// §6.8 ST step skeleton. One M_Step per step, one commit via M_Advance.
METHOD M_ChainRun
IF NOT _attached THEN
    RETURN;
END_IF
CASE _step OF
    0:  // ram up
        M_Step(StepNo := _baseStepNo, StepName := 'project.step.pressSafePositionRamUp',
            Awaits := _pressRam, AwaitingLabel := 'PressRam.RETRACT',
            TimeClass := E_TimeClass.WORK, ExpectedTime := T#0S, Branch := 0);
        IF M_TryIssue(Steppable := TRUE) THEN
            _pressRam.Abort := FALSE;
            _pressRam.Command := E_CylinderCommand.RETRACT;
            _pressRam.Execute := TRUE;
        END_IF
        IF _pressRam.Done THEN
            _pressRam.Execute := FALSE;
            _retVal := E_StepResult.ADVANCE;
        END_IF
        M_Advance(OnAdvance := 20, OnJump1 := -1, OnJump2 := -1, OnJump3 := -1);
    20:  // door open
        M_Step(StepNo := _baseStepNo + 20, StepName := 'project.step.pressSafePositionDoorOpen',
            Awaits := _door, AwaitingLabel := 'Door.RETRACT',
            TimeClass := E_TimeClass.WORK, ExpectedTime := T#0S, Branch := 0);
        IF M_TryIssue(Steppable := TRUE) THEN
            _door.Abort := FALSE;
            _door.Command := E_CylinderCommand.RETRACT;
            _door.Execute := TRUE;
        END_IF
        IF _door.Done THEN
            _door.Execute := FALSE;
            _retVal := E_StepResult.ADVANCE;
        END_IF
        M_Advance(OnAdvance := 40, OnJump1 := -1, OnJump2 := -1, OnJump3 := -1);
    40:  // slide outside
        M_Step(StepNo := _baseStepNo + 40, StepName := 'project.step.pressSafePositionSlideOutside',
            Awaits := _partSlide, AwaitingLabel := 'PartSlide.RETRACT',
            TimeClass := E_TimeClass.WORK, ExpectedTime := T#0S, Branch := 0);
        IF M_TryIssue(Steppable := TRUE) THEN
            _partSlide.Abort := FALSE;
            _partSlide.Command := E_CylinderCommand.RETRACT;
            _partSlide.Execute := TRUE;
        END_IF
        IF _partSlide.Done THEN
            _partSlide.Execute := FALSE;
            _retVal := E_StepResult.ADVANCE;
        END_IF
        M_Advance(OnAdvance := 999, OnJump1 := -1, OnJump2 := -1, OnJump3 := -1);
    999:  // established
        M_Step(StepNo := _baseStepNo + 60, StepName := 'project.step.pressSafePositionComplete',
            Awaits := 0, AwaitingLabel := '', TimeClass := E_TimeClass.WORK, ExpectedTime := T#0S, Branch := 0);
        Done := TRUE;
ELSE
    M_Fault(Reason := E_Reason.STEP_STALLED, DescriptionKey := 'std.error.undefinedStep');
END_CASE
END_METHOD

METHOD Setup : BOOL
VAR_INPUT
    Host : I_SequenceHost;
END_VAR
VAR_IN_OUT
    PressRam : FB_CylinderCM;
    Door : FB_CylinderCM;
    PartSlide : FB_CylinderCM;
END_VAR
_pressRam REF= PressRam;
_door REF= Door;
_partSlide REF= PartSlide;
Setup := M_Attach(Host := Host)
    AND __ISVALIDREF(_pressRam) AND __ISVALIDREF(_door) AND __ISVALIDREF(_partSlide);
END_METHOD

END_FUNCTION_BLOCK

// ---- 01_PneumaticPress/Sequences/FB_PressDemoChangeover.TcPOU
// CHANGEOVER mode chain (Core §6.2/§6.8 ST skeleton on FB_SequenceBase): validate
// the selected model, establish the shared load-safe position, then ask the
// operator (§6.11) to confirm tooling/material match before completing. The
// 'repeat position' answer restarts the guided move via a backward jump (§6.10).
FUNCTION_BLOCK FB_PressDemoChangeover EXTENDS FB_SequenceBase
VAR
    _decisionRequest : ST_DecisionRequest;
    _answer : INT;
    _modelSelected : BOOL;
    {attribute 'OPC.UA.DA' := '0'}
    _outCmd : REFERENCE TO ST_PneumaticPressOutCmd;
    {attribute 'OPC.UA.DA' := '0'}
    _model : REFERENCE TO ST_ModelId;
    {attribute 'OPC.UA.DA' := '0'}
    _loadPosition : FB_PressDemoLoadPosition;
END_VAR

// §6.8 - the chain's own state on a restart (the base resets the flow state).
METHOD PROTECTED OnChainReset
_answer := 0;
END_METHOD

METHOD M_Run
IF NOT _attached THEN
    RETURN;
END_IF
CASE _step OF
    0:  // initialize
        M_Step(StepNo := 0, StepName := 'project.step.pressChangeoverInitialize',
            Awaits := 0, AwaitingLabel := '', TimeClass := E_TimeClass.WORK, ExpectedTime := T#0S, Branch := 0);
        _outCmd.ChangeoverCompleted := FALSE;
        _answer := 0;
        _decisionRequest.Prompt := '';
        M_ClearDecision();
        _retVal := E_StepResult.ADVANCE;
        M_Advance(OnAdvance := 800, OnJump1 := -1, OnJump2 := -1, OnJump3 := -1);
    800:  // validate the transactionally-loaded model
        M_Step(StepNo := 800, StepName := 'project.step.pressChangeoverValidateModel',
            Awaits := 0, AwaitingLabel := '', TimeClass := E_TimeClass.WAIT_OPERATOR, ExpectedTime := T#0S, Branch := 0);
        _modelSelected := M_Await(Idx := 1, Label := 'project.condition.pressModelSelected',
            Ok := _model.ModelCode <> '');
        IF _modelSelected THEN
            _retVal := E_StepResult.ADVANCE;
        END_IF
        M_Advance(OnAdvance := 810, OnJump1 := -1, OnJump2 := -1, OnJump3 := -1);
    810:  // shared load-safe position (composite step)
        _retVal := M_RunSub(Chain := _loadPosition, BaseStepNo := 810);
        M_Advance(OnAdvance := 870, OnJump1 := -1, OnJump2 := -1, OnJump3 := -1);
    870:  // request tooling/material confirmation
        M_Step(StepNo := 870, StepName := 'project.step.pressChangeoverRequestConfirmation',
            Awaits := 0, AwaitingLabel := '', TimeClass := E_TimeClass.WAIT_OPERATOR, ExpectedTime := T#0S, Branch := 0);
        _decisionRequest.Prompt := 'project.decision.pressChangeoverConfirm';
        _decisionRequest.Options[1] := 'project.decision.confirmChangeover';
        _decisionRequest.Options[2] := 'project.decision.repeatChangeoverPosition';
        _decisionRequest.Default := 0;
        _decisionRequest.Timeout := T#0S;
        M_AskDecision(Req := _decisionRequest);
        _retVal := E_StepResult.ADVANCE;
        M_Advance(OnAdvance := 880, OnJump1 := -1, OnJump2 := -1, OnJump3 := -1);
    880:  // await confirmation; JUMP1 = repeat the guided position
        M_Step(StepNo := 880, StepName := 'project.step.pressChangeoverAwaitConfirmation',
            Awaits := 0, AwaitingLabel := '', TimeClass := E_TimeClass.WAIT_OPERATOR, ExpectedTime := T#0S, Branch := 0);
        _answer := M_TakeDecision();
        IF _answer = 1 THEN
            _retVal := E_StepResult.ADVANCE;
        ELSIF _answer = 2 THEN
            _retVal := E_StepResult.JUMP1;
        ELSE
            _modelSelected := M_Await(Idx := 1,
                Label := 'project.condition.pressChangeoverConfirmation', Ok := FALSE);
        END_IF
        M_Advance(OnAdvance := 999, OnJump1 := 810, OnJump2 := -1, OnJump3 := -1);
    999:  // complete
        M_Step(StepNo := 999, StepName := 'project.step.pressChangeoverComplete',
            Awaits := 0, AwaitingLabel := '', TimeClass := E_TimeClass.WORK, ExpectedTime := T#0S, Branch := 0);
        _outCmd.ChangeoverCompleted := TRUE;
        M_Complete();
ELSE
    M_Fault(Reason := E_Reason.STEP_STALLED, DescriptionKey := 'std.error.undefinedStep');
END_CASE
END_METHOD

METHOD Setup : BOOL
VAR_INPUT
    Host : I_SequenceHost;
END_VAR
VAR_IN_OUT
    PressRam : FB_CylinderCM;
    Door : FB_CylinderCM;
    PartSlide : FB_CylinderCM;
    OutCmd : ST_PneumaticPressOutCmd;
    Model : ST_ModelId;
END_VAR
_outCmd REF= OutCmd;
_model REF= Model;
Setup := M_Attach(Host := Host) AND __ISVALIDREF(_outCmd) AND __ISVALIDREF(_model)
    AND _loadPosition.Setup(Host := Host, PressRam := PressRam, Door := Door, PartSlide := PartSlide);
END_METHOD

END_FUNCTION_BLOCK

// ---- 01_PneumaticPress/Sequences/FB_PressDemoAuto.TcPOU
// AUTO mode chain (Core §6.2/§6.8 ST skeleton on FB_SequenceBase): the continuous
// production cycle — await a fresh two-hand start with part+air present, transfer
// the part in, press for the recipe dwell, return to load position, count the good
// part, and loop until Stop. A Stop requested at the between-cycles wait is honored
// there (M_StopNow) so no phantom cycle is charged. Every child motion goes through
// the §6.1 handshake (M_TryIssue); progression rides the shared _retVal.
FUNCTION_BLOCK FB_PressDemoAuto EXTENDS FB_SequenceBase
VAR
    _partReady, _airReady, _startReady : BOOL;
    _dwellTwoHandHeld : BOOL;          // N220 named wait: two-hand held through the dwell
    _decisionRequest : ST_DecisionRequest;   // §6.11 not-reached confirmation
    _answer : INT;
    _ramReached, _failureConfirmed : BOOL;   // N200/N210 named waits
    _twoHandHeldDuringClose : BOOL;          // N180 named wait
    _closeAbortWarned : BOOL;                // N180 §6.9(e) message result
    _ramFailureReported : BOOL;              // N200 §6.9(e) message result
    _partInMachine : BOOL;                   // §3.16.3 the part is already received
    _partDispositioned : BOOL;               // N260 already set the verdict
    _traceAccepted, _recordAccepted, _partProcessed : BOOL;
    {attribute 'OPC.UA.DA' := '0'}
    _pressRam : REFERENCE TO FB_CylinderCM;
    {attribute 'OPC.UA.DA' := '0'}
    _door : REFERENCE TO FB_CylinderCM;
    {attribute 'OPC.UA.DA' := '0'}
    _partSlide : REFERENCE TO FB_CylinderCM;
    {attribute 'OPC.UA.DA' := '0'}
    _twoHand : REFERENCE TO FB_TwoHandStartCM;
    {attribute 'OPC.UA.DA' := '0'}
    _partPresentSensor : REFERENCE TO FB_DigitalInputCM;
    {attribute 'OPC.UA.DA' := '0'}
    _airPressureMonitor : REFERENCE TO FB_AirPressureMonitorCM;
    {attribute 'OPC.UA.DA' := '0'}
    _parCfg : REFERENCE TO ST_PneumaticPressParCfg;
    // §3.8a - the CELL's own policy, held separately from the MODEL's data and
    // referenced exactly like _parCfg, so each step reads whichever structure
    // actually owns the value it is asking about.
    {attribute 'OPC.UA.DA' := '0'}
    _stationCfg : REFERENCE TO ST_PneumaticPressStationCfg;
    {attribute 'OPC.UA.DA' := '0'}
    _outCmd : REFERENCE TO ST_PneumaticPressOutCmd;
    {attribute 'OPC.UA.DA' := '0'}
    _startLatched : REFERENCE TO BOOL;
    {attribute 'OPC.UA.DA' := '0'}
    _loadPosition : FB_PressDemoLoadPosition;
END_VAR

// §6.8 - the chain's own state on a restart (the base resets the flow state).
METHOD PROTECTED OnChainReset
// A chart restart abandons whatever the cycle was holding: the part record is
// closed by N215/N999, never by a restart, so both trackers start clean.
_partDispositioned := FALSE;
_partInMachine := FALSE;
END_METHOD

METHOD M_Run
IF NOT _attached THEN
    RETURN;
END_IF
CASE _step OF
    0:  // initialize
        M_Step(StepNo := 0, StepName := 'project.step.pressAutoInitialize',
            Awaits := 0, AwaitingLabel := '', TimeClass := E_TimeClass.WORK, ExpectedTime := T#0S, Branch := 0);
        _outCmd.CycleCompleted := FALSE;
        _retVal := E_StepResult.ADVANCE;
        M_Advance(OnAdvance := 100, OnJump1 := -1, OnJump2 := -1, OnJump3 := -1 );
    100:  // await a fresh two-hand start (the §8.11.1 cycle-start marker)
        M_Step(StepNo := 100, StepName := 'project.step.pressAwaitTwoHand',
            Awaits := 0, AwaitingLabel := '', TimeClass := E_TimeClass.WAIT_OPERATOR, ExpectedTime := T#0S, Branch := 0);
        _outCmd.CycleCompleted := FALSE;
        _partReady := M_Await(Idx := 1, Label := 'project.condition.partPresent',
            Ok := _partPresentSensor.OutImm.Value AND _partPresentSensor.OutImm.Quality);
        _airReady := M_Await(Idx := 2, Label := 'project.condition.airPressureOk',
            Ok := _airPressureMonitor.OutImm.PressureOk);
        IF _stationCfg.RequireTwoHandStart THEN
            _startReady := M_Await(Idx := 3, Label := 'project.condition.twoHandStart', Ok := _startLatched);
        ELSE
            _startReady := TRUE;
        END_IF
        IF M_StopPending() THEN
            M_StopNow();                       // stop accepted BETWEEN cycles: no phantom cycle
        ELSIF _partReady AND _airReady AND _startReady THEN
            // §3.16.3 receive once per PHYSICAL part. The N180 two-hand abort returns
            // here with the same part still in the machine and nothing processed, so a
            // second M_PartReceived would open a duplicate record for one part.
            // M_PartStarted (N150) is deliberately NOT guarded: each pass is a genuine
            // processing attempt on that part.
            IF NOT _partInMachine THEN
                _traceAccepted := M_PartReceived();
                _partInMachine := TRUE;
            END_IF
            _retVal := E_StepResult.ADVANCE;
        END_IF
        M_Advance(OnAdvance := 110, OnJump1 := -1, OnJump2 := -1, OnJump3 := -1);
    110:  // ram up
        M_Step(StepNo := 110, StepName := 'project.step.pressRamUp',
            Awaits := _pressRam, AwaitingLabel := 'PressRam.RETRACT', TimeClass := E_TimeClass.WORK, ExpectedTime := T#0S, Branch := 0);
        IF M_TryIssue(Steppable := TRUE) THEN
            _pressRam.Abort := FALSE; _pressRam.Command := E_CylinderCommand.RETRACT; _pressRam.Execute := TRUE;
        END_IF
        IF _pressRam.Done THEN _pressRam.Execute := FALSE; _retVal := E_StepResult.ADVANCE; END_IF
        M_Advance(OnAdvance := 130, OnJump1 := -1, OnJump2 := -1, OnJump3 := -1);
    130:  // door open
        M_Step(StepNo := 130, StepName := 'project.step.pressDoorOpen',
            Awaits := _door, AwaitingLabel := 'Door.RETRACT', TimeClass := E_TimeClass.WORK, ExpectedTime := T#0S, Branch := 0);
        IF M_TryIssue(Steppable := TRUE) THEN
            _door.Abort := FALSE; _door.Command := E_CylinderCommand.RETRACT; _door.Execute := TRUE;
        END_IF
        IF _door.Done THEN _door.Execute := FALSE; _retVal := E_StepResult.ADVANCE; END_IF
        M_Advance(OnAdvance := 150, OnJump1 := -1, OnJump2 := -1, OnJump3 := -1);
    150:  // slide inside (value-adding sequence begins)
        M_Step(StepNo := 150, StepName := 'project.step.pressSlideInside',
            Awaits := _partSlide, AwaitingLabel := 'PartSlide.EXTEND', TimeClass := E_TimeClass.WORK, ExpectedTime := T#0S, Branch := 0);
        IF M_TryIssue(Steppable := TRUE) THEN
            M_PartStarted();
            _partSlide.Abort := FALSE; _partSlide.Command := E_CylinderCommand.EXTEND; _partSlide.Execute := TRUE;
        END_IF
        IF _partSlide.Done THEN _partSlide.Execute := FALSE; _retVal := E_StepResult.ADVANCE; END_IF
        M_Advance(OnAdvance := 170, OnJump1 := -1, OnJump2 := -1, OnJump3 := -1);
    170:  // transfer settle
        M_Step(StepNo := 170, StepName := 'project.step.pressTransferSettle',
            Awaits := 0, AwaitingLabel := '', TimeClass := E_TimeClass.WORK, ExpectedTime := _parCfg.TransferSettleTime, Branch := 0);
        _retVal := M_Delay(PT := _parCfg.TransferSettleTime);
        M_Advance(OnAdvance := 180, OnJump1 := -1, OnJump2 := -1, OnJump3 := -1);
    180:  // door close. Releasing a two-hand button while the door is moving is an
          // operator abort, not a fault: the door goes back up, the part slides out,
          // and the cycle returns to the two-hand wait (§6.10 jump). Completion wins
          // if the door finished in the same scan the button was released.
        M_Step(StepNo := 180, StepName := 'project.step.pressDoorClose',
            Awaits := _door, AwaitingLabel := 'Door.EXTEND', TimeClass := E_TimeClass.WORK, ExpectedTime := T#0S, Branch := 0);
        _twoHandHeldDuringClose := M_Await(Idx := 1,
            Label := 'project.condition.twoHandHeldDuringDoorClose',
            Ok := _twoHand.OutImm.SafeActive OR NOT _stationCfg.RequireTwoHandStart);
        IF M_TryIssue(Steppable := TRUE) THEN
            _door.Abort := FALSE; _door.Command := E_CylinderCommand.EXTEND; _door.Execute := TRUE;
        END_IF
        IF _door.Done THEN
            _door.Execute := FALSE;
            _retVal := E_StepResult.ADVANCE;
        ELSIF NOT _twoHandHeldDuringClose THEN
            _door.Execute := FALSE;             // §6.1 Execute-drop reset releases the close
            // §6.9(e) — a WARNING, not a fault: the release is designed operator
            // behaviour and the chain already owns the recovery below, so nothing
            // stops. It is recorded because a cycle was abandoned with the part
            // still in the machine, and the §3.13 chart marks this step for it.
            // The base raises it once per visit however many scans this runs.
            _closeAbortWarned := M_RaiseWarning(
                Reason := PL_PressReasons.PRESS_TWO_HAND_RELEASED,
                DescriptionKey := 'project.warning.twoHandReleasedDuringDoorClose',
                Severity := E_Severity.LOW, Category := E_Category.PROCESS);
            _retVal := E_StepResult.JUMP1;      // released -> reopen and clear the part
        END_IF
        M_Advance(OnAdvance := 200, OnJump1 := 185, OnJump2 := -1, OnJump3 := -1);
    185:  // two-hand released during closing: take the door back up
        M_Step(StepNo := 185, StepName := 'project.step.pressDoorReopen',
            Awaits := _door, AwaitingLabel := 'Door.RETRACT', TimeClass := E_TimeClass.WORK, ExpectedTime := T#0S, Branch := 0);
        IF M_TryIssue(Steppable := TRUE) THEN
            _door.Abort := FALSE; _door.Command := E_CylinderCommand.RETRACT; _door.Execute := TRUE;
        END_IF
        IF _door.Done THEN _door.Execute := FALSE; _retVal := E_StepResult.ADVANCE; END_IF
        M_Advance(OnAdvance := 190, OnJump1 := -1, OnJump2 := -1, OnJump3 := -1);
    190:  // slide the part back out, then return to the two-hand wait. The start latch
          // is dropped so the cycle cannot resume without a fresh two-hand press.
        M_Step(StepNo := 190, StepName := 'project.step.pressSlideOutsideAfterAbort',
            Awaits := _partSlide, AwaitingLabel := 'PartSlide.RETRACT', TimeClass := E_TimeClass.WORK, ExpectedTime := T#0S, Branch := 0);
        IF M_TryIssue(Steppable := TRUE) THEN
            _partSlide.Abort := FALSE; _partSlide.Command := E_CylinderCommand.RETRACT; _partSlide.Execute := TRUE;
        END_IF
        IF _partSlide.Done THEN
            _partSlide.Execute := FALSE;
            _startLatched := FALSE;
            _retVal := E_StepResult.ADVANCE;
        END_IF
        M_Advance(OnAdvance := 100, OnJump1 := -1, OnJump2 := -1, OnJump3 := -1);
    200:  // ram down. THIS step owns the not-reached disposition, so it does NOT hand
          // the ram to the §6.9 auto-rollup: an awaited child fault is adopted by the
          // Unit (ERROR, _step := 0) before _M_Dispatch runs, and the chain would stop
          // before it could ask the operator anything. The wait is still named (§6.9(b))
          // and the cylinder still raises its own CYL_NOT_EXTENDED alarm.
        M_Step(StepNo := 200, StepName := 'project.step.pressRamDown',
            Awaits := 0, AwaitingLabel := '', TimeClass := E_TimeClass.WORK, ExpectedTime := T#0S, Branch := 0);
        _ramReached := M_Await(Idx := 1, Label := 'project.condition.pressRamExtended',
            Ok := _pressRam.Done);
        IF M_TryIssue(Steppable := TRUE) THEN
            _pressRam.Abort := FALSE; _pressRam.Command := E_CylinderCommand.EXTEND; _pressRam.Execute := TRUE;
        END_IF
        IF _pressRam.Done THEN
            _pressRam.Execute := FALSE;
            _retVal := E_StepResult.ADVANCE;
        ELSIF _pressRam.Error THEN
            // §6.9(e) — publish the ram's own first-out (CYL_NOT_EXTENDED, with its
            // text and IO tag) on the Unit and on this row of the §3.13 chart, and
            // do NOT adopt it: the confirmation + scrap below IS the handling, so a
            // fault here would replace a designed recovery. Saying nothing is what
            // left the failure visible only on the ram itself.
            _ramFailureReported := M_ReportFromChild(Source := _pressRam);
            _pressRam.Execute := FALSE;         // §6.1 Execute-drop reset returns the ram to READY
            _retVal := E_StepResult.JUMP1;      // did not reach -> operator confirmation
        END_IF
        M_Advance(OnAdvance := 220, OnJump1 := 210, OnJump2 := -1, OnJump3 := -1);
    210:  // press did not reach: the operator confirms the failure before the part is
          // scrapped. A scrap is deliberate, so there is no timeout default (§6.11).
        M_Step(StepNo := 210, StepName := 'project.step.pressNotReachedConfirm',
            Awaits := 0, AwaitingLabel := '', TimeClass := E_TimeClass.WAIT_OPERATOR, ExpectedTime := T#0S, Branch := 0);
        _decisionRequest.Prompt := 'project.decision.pressNotReached';
        _decisionRequest.Options[1] := 'project.decision.confirmScrapAndReturn';
        _decisionRequest.Default := 0;
        _decisionRequest.Timeout := T#0S;
        M_AskDecision(Req := _decisionRequest);
        _answer := M_TakeDecision();
        IF _answer = 1 THEN
            _retVal := E_StepResult.ADVANCE;
        ELSE
            _failureConfirmed := M_Await(Idx := 1,
                Label := 'project.condition.pressFailureConfirmation', Ok := FALSE);
        END_IF
        M_Advance(OnAdvance := 215, OnJump1 := -1, OnJump2 := -1, OnJump3 := -1);
    215:  // disposition the part NOK, then rejoin the shared return-to-start step
        M_Step(StepNo := 215, StepName := 'project.step.pressScrapPart',
            Awaits := 0, AwaitingLabel := '', TimeClass := E_TimeClass.WORK, ExpectedTime := T#0S, Branch := 0);
        _partProcessed := M_PartProcessed(Verdict := E_Verdict.NOK,
            Reason := PL_ModuleReasons.CYL_NOT_EXTENDED);
        _partDispositioned := TRUE;             // N999 must not also count it good
        _partInMachine := FALSE;                // dispositioned: the next one is a new part
        _outCmd.CycleCompleted := FALSE;
        _retVal := E_StepResult.ADVANCE;
        M_Advance(OnAdvance := 240, OnJump1 := -1, OnJump2 := -1, OnJump3 := -1);
    220:  // press dwell — two-hand must stay held; releasing it HOLDS the dwell
        M_Step(StepNo := 220, StepName := 'project.step.pressDwell',
            Awaits := 0, AwaitingLabel := '', TimeClass := E_TimeClass.WORK, ExpectedTime := _parCfg.PressSettleTime, Branch := 0);
        // Releasing the button mid-dwell is the designed way to stop pressing, so it
        // is a named wait (§6.9(b)), not a fault: the ram's outputs come off, the
        // dwell timer freezes where it is because M_Delay is not called, and pressing
        // again restores the force and finishes the remaining dwell. Faulting here
        // charged an unrecoverable downtime event for normal operator behaviour.
        _dwellTwoHandHeld := M_Await(Idx := 1, Label := 'project.condition.twoHandHeldDuringPress',
            Ok := _twoHand.OutImm.SafeActive OR NOT _stationCfg.RequireTwoHandStart);
        IF NOT _dwellTwoHandHeld THEN
            _pressRam.WithdrawOutputs();
        ELSE
            // The press force is the valve latched by the EXTEND that step 200 already
            // completed, so after a withdraw only this call re-energizes it — and the
            // ram re-checks its own extend permit before it does (§7.2).
            _pressRam.RestoreOutputs();
            _retVal := M_Delay(PT := _parCfg.PressSettleTime);
        END_IF
        M_Advance(OnAdvance := 230, OnJump1 := -1, OnJump2 := -1, OnJump3 := -1);
    230:  // record the applied dwell (§3.16.1 measured value)
        M_Step(StepNo := 230, StepName := 'project.step.pressRecordResult',
            Awaits := 0, AwaitingLabel := '', TimeClass := E_TimeClass.WORK, ExpectedTime := T#0S, Branch := 0);
        _recordAccepted := M_PartRecord(RecordName := 'PressDwell',
            Value := DINT_TO_LREAL(TIME_TO_DINT(_parCfg.PressSettleTime)),
            Minimum := 0, Maximum := 30000,
            Target := DINT_TO_LREAL(TIME_TO_DINT(_parCfg.PressSettleTime)), EngUnit := 'ms');
        _retVal := E_StepResult.ADVANCE;
        M_Advance(OnAdvance := 240, OnJump1 := -1, OnJump2 := -1, OnJump3 := -1);
    240:  // return to the shared load-safe position (composite step)
        _retVal := M_RunSub(Chain := _loadPosition, BaseStepNo := 240);
        M_Advance(OnAdvance := 999, OnJump1 := -1, OnJump2 := -1, OnJump3 := -1);
    999:  // cycle complete — write result, count by verdict, loop (§8.11.1 finish marker)
        M_Step(StepNo := 999, StepName := 'project.step.pressAutoComplete',
            Awaits := 0, AwaitingLabel := '', TimeClass := E_TimeClass.WORK, ExpectedTime := T#0S, Branch := 0);
        _outCmd.CycleCompleted := TRUE;
        IF _partDispositioned THEN
            _partDispositioned := FALSE;       // N260 already set the NOK verdict
        ELSE
            _partProcessed := M_PartProcessed(Verdict := E_Verdict.OK, Reason := E_Reason.NONE);
            IF NOT _partProcessed THEN
                M_CountGood();                 // §3.9: no carrier configured — count directly
            END_IF
        END_IF
        _partInMachine := FALSE;               // processed: the next one is a new part
        _startLatched := FALSE;
        IF M_EndOfCycle() THEN
            _retVal := E_StepResult.ADVANCE;   // stop NOT requested: loop to N100
        END_IF
        M_Advance(OnAdvance := 100, OnJump1 := -1, OnJump2 := -1, OnJump3 := -1);
ELSE
    M_Fault(Reason := E_Reason.STEP_STALLED, DescriptionKey := 'std.error.undefinedStep');
END_CASE
END_METHOD

METHOD Setup : BOOL
VAR_INPUT
    Host : I_SequenceHost;
END_VAR
VAR_IN_OUT
    PressRam : FB_CylinderCM;
    Door : FB_CylinderCM;
    PartSlide : FB_CylinderCM;
    TwoHand : FB_TwoHandStartCM;
    PartPresentSensor : FB_DigitalInputCM;
    AirPressureMonitor : FB_AirPressureMonitorCM;
    ParCfg : ST_PneumaticPressParCfg;
    StationCfg : ST_PneumaticPressStationCfg;
    OutCmd : ST_PneumaticPressOutCmd;
    StartLatched : BOOL;
END_VAR
_pressRam REF= PressRam;
_door REF= Door;
_partSlide REF= PartSlide;
_twoHand REF= TwoHand;
_partPresentSensor REF= PartPresentSensor;
_airPressureMonitor REF= AirPressureMonitor;
_parCfg REF= ParCfg;
_stationCfg REF= StationCfg;
_outCmd REF= OutCmd;
_startLatched REF= StartLatched;
Setup := M_Attach(Host := Host) AND __ISVALIDREF(_pressRam) AND __ISVALIDREF(_door)
    AND __ISVALIDREF(_partSlide) AND __ISVALIDREF(_twoHand)
    AND __ISVALIDREF(_partPresentSensor) AND __ISVALIDREF(_airPressureMonitor)
    AND __ISVALIDREF(_parCfg) AND __ISVALIDREF(_outCmd) AND __ISVALIDREF(_startLatched)
    AND _loadPosition.Setup(Host := Host, PressRam := PressRam, Door := Door, PartSlide := PartSlide);
END_METHOD

END_FUNCTION_BLOCK

// ---- 01_PneumaticPress/Sequences/FB_SFC_PressDemoAuto.TcPOU
// SFC rendition of FB_PressDemoAuto - identical behaviour, chart-language
// transitions. Every step action below sets the shared `_retVal`; the chart's
// transitions read it, and the owner calls M_BeginScan() once per PLC cycle
// before executing this chart so the result cannot survive into the next scan
// (Core §6.8). The ST twin remains FB_PressDemoAuto; keep the two in step.
FUNCTION_BLOCK INTERNAL FB_SFC_PressDemoAuto EXTENDS FB_SequenceBase
VAR
    _partReady, _airReady, _startReady : BOOL;
    _dwellTwoHandHeld : BOOL;          // N220 named wait: two-hand held through the dwell
    _decisionRequest : ST_DecisionRequest;   // §6.11 not-reached confirmation
    _answer : INT;
    _ramReached, _failureConfirmed : BOOL;   // N200/N210 named waits
    _twoHandHeldDuringClose : BOOL;
    _closeAbortWarned : BOOL;                // N180 §6.9(e) message result
    _ramFailureReported : BOOL;              // N200 §6.9(e) message result          // N180 named wait
    _partInMachine : BOOL;                   // §3.16.3 the part is already received
    _partDispositioned : BOOL;               // N260 already set the verdict
    _traceAccepted, _recordAccepted, _partProcessed : BOOL;
    {attribute 'OPC.UA.DA' := '0'}
    _pressRam : REFERENCE TO FB_CylinderCM;
    {attribute 'OPC.UA.DA' := '0'}
    _door : REFERENCE TO FB_CylinderCM;
    {attribute 'OPC.UA.DA' := '0'}
    _partSlide : REFERENCE TO FB_CylinderCM;
    {attribute 'OPC.UA.DA' := '0'}
    _twoHand : REFERENCE TO FB_TwoHandStartCM;
    {attribute 'OPC.UA.DA' := '0'}
    _partPresentSensor : REFERENCE TO FB_DigitalInputCM;
    {attribute 'OPC.UA.DA' := '0'}
    _airPressureMonitor : REFERENCE TO FB_AirPressureMonitorCM;
    {attribute 'OPC.UA.DA' := '0'}
    _parCfg : REFERENCE TO ST_PneumaticPressParCfg;
    // §3.8a - the CELL's own policy, held separately from the MODEL's data and
    // referenced exactly like _parCfg, so each step reads whichever structure
    // actually owns the value it is asking about.
    {attribute 'OPC.UA.DA' := '0'}
    _stationCfg : REFERENCE TO ST_PneumaticPressStationCfg;
    {attribute 'OPC.UA.DA' := '0'}
    _outCmd : REFERENCE TO ST_PneumaticPressOutCmd;
    {attribute 'OPC.UA.DA' := '0'}
    _startLatched : REFERENCE TO BOOL;
    {attribute 'OPC.UA.DA' := '0'}
    _loadPosition : FB_PressDemoLoadPosition;
END_VAR

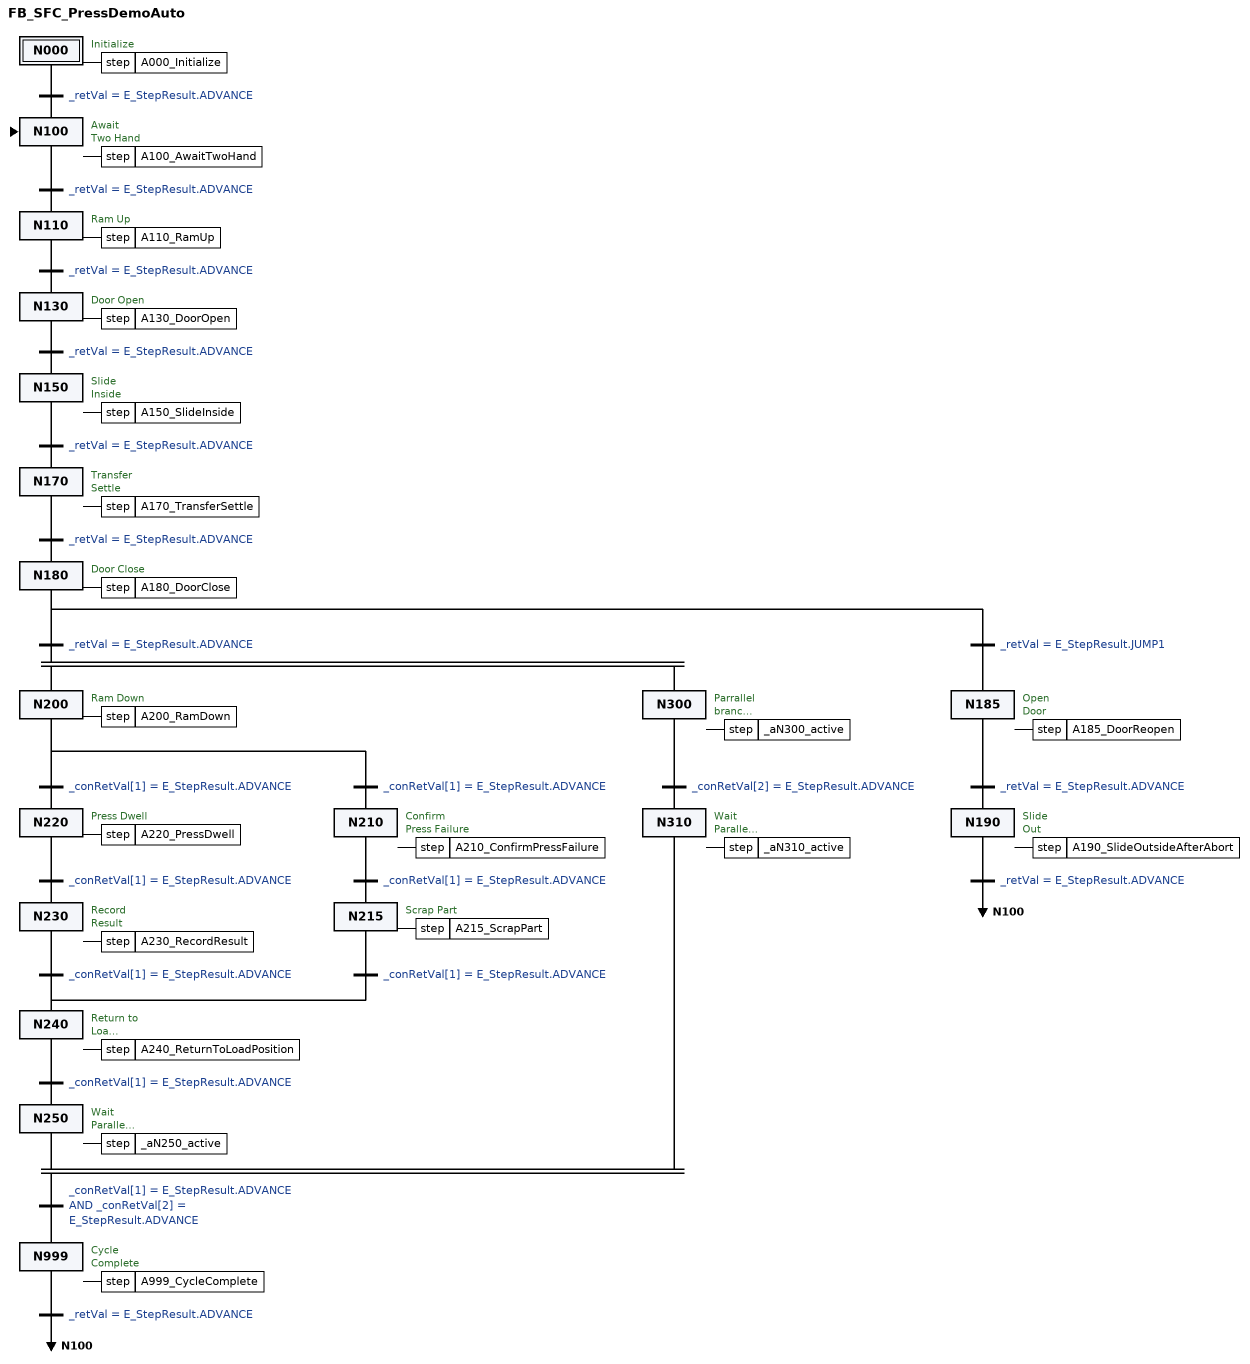
// Initialize
INITIAL_STEP N000:
    A000_Initialize(N);  // step action
END_STEP
TRANSITION FROM N000 TO N100
    := _retVal = E_StepResult.ADVANCE;
END_TRANSITION
// Await
// Two Hand
STEP N100:
    A100_AwaitTwoHand(N);  // step action
END_STEP
TRANSITION FROM N100 TO N110
    := _retVal = E_StepResult.ADVANCE;
END_TRANSITION
// Ram Up
STEP N110:
    A110_RamUp(N);  // step action
END_STEP
TRANSITION FROM N110 TO N130
    := _retVal = E_StepResult.ADVANCE;
END_TRANSITION
// Door Open
STEP N130:
    A130_DoorOpen(N);  // step action
END_STEP
TRANSITION FROM N130 TO N150
    := _retVal = E_StepResult.ADVANCE;
END_TRANSITION
// Slide
// Inside
STEP N150:
    A150_SlideInside(N);  // step action
END_STEP
TRANSITION FROM N150 TO N170
    := _retVal = E_StepResult.ADVANCE;
END_TRANSITION
// Transfer
// Settle
STEP N170:
    A170_TransferSettle(N);  // step action
END_STEP
TRANSITION FROM N170 TO N180
    := _retVal = E_StepResult.ADVANCE;
END_TRANSITION
// Door Close
STEP N180:
    A180_DoorClose(N);  // step action
END_STEP
TRANSITION FROM N180 TO (N200, N300)
    := _retVal = E_StepResult.ADVANCE;
END_TRANSITION
// Ram Down
STEP N200:
    A200_RamDown(N);  // step action
END_STEP
TRANSITION FROM N200 TO N220
    := _conRetVal[1] = E_StepResult.ADVANCE;
END_TRANSITION
// Press Dwell
STEP N220:
    A220_PressDwell(N);  // step action
END_STEP
TRANSITION FROM N220 TO N230
    := _conRetVal[1] = E_StepResult.ADVANCE;
END_TRANSITION
// Record
// Result
STEP N230:
    A230_RecordResult(N);  // step action
END_STEP
TRANSITION FROM N230 TO N240
    := _conRetVal[1] = E_StepResult.ADVANCE;
END_TRANSITION
TRANSITION FROM N200 TO N210
    := _conRetVal[1] = E_StepResult.ADVANCE;
END_TRANSITION
// Confirm
// Press Failure
STEP N210:
    A210_ConfirmPressFailure(N);  // step action
END_STEP
TRANSITION FROM N210 TO N215
    := _conRetVal[1] = E_StepResult.ADVANCE;
END_TRANSITION
// Scrap Part
STEP N215:
    A215_ScrapPart(N);  // step action
END_STEP
TRANSITION FROM N215 TO N240
    := _conRetVal[1] = E_StepResult.ADVANCE;
END_TRANSITION
// Return to
// Load
// Position
STEP N240:
    A240_ReturnToLoadPosition(N);  // step action
END_STEP
TRANSITION FROM N240 TO N250
    := _conRetVal[1] = E_StepResult.ADVANCE;
END_TRANSITION
// Wait
// Parallel
// Branch
STEP N250:
    _aN250_active(N);  // step action
END_STEP
// Parrallel
// branch
// example
STEP N300:
    _aN300_active(N);  // step action
END_STEP
TRANSITION FROM N300 TO N310
    := _conRetVal[2] = E_StepResult.ADVANCE;
END_TRANSITION
// Wait
// Parallel
// Branch
STEP N310:
    _aN310_active(N);  // step action
END_STEP
TRANSITION FROM N180 TO N185
    := _retVal = E_StepResult.JUMP1;
END_TRANSITION
// Open
// Door
STEP N185:
    A185_DoorReopen(N);  // step action
END_STEP
TRANSITION FROM N185 TO N190
    := _retVal = E_StepResult.ADVANCE;
END_TRANSITION
// Slide
// Out
STEP N190:
    A190_SlideOutsideAfterAbort(N);  // step action
END_STEP
TRANSITION FROM N190 TO N100
    := _retVal = E_StepResult.ADVANCE;
END_TRANSITION
TRANSITION FROM (N250, N310) TO N999
    := _conRetVal[1] = E_StepResult.ADVANCE AND _conRetVal[2] = E_StepResult.ADVANCE;
END_TRANSITION
// Cycle
// Complete
STEP N999:
    A999_CycleComplete(N);  // step action
END_STEP
TRANSITION FROM N999 TO N100
    := _retVal = E_StepResult.ADVANCE;
END_TRANSITION

ACTION _aN250_active:
// N250 — leg 1 waits at the join. §6.12: the parallel divergence after A180 is
// drawn INSIDE this POU, so both legs share the FB and each leg step says which leg
// it is through `Branch` on its own step record - a leg can never be declared
// without recording a step.
//
// NEITHER leg is the main line. A simultaneous divergence has N equal legs, so
// numbering one of them 0 would have made it look subordinate on the §3.13 chart
// and left `_retVal` meaning two different things depending on where you were
// reading it. `_retVal` is the single-threaded line before and after the fork;
// inside it, leg 1 is `_conRetVal[1]` and leg 2 is `_conRetVal[2]`.
M_Step(StepNo := 250, StepName := 'project.step.pressAwaitParallelBranch', Awaits := 0,
    AwaitingLabel := '', TimeClass := E_TimeClass.WORK, ExpectedTime := T#0S,
    Branch := 1);
_conRetVal[1] := E_StepResult.ADVANCE;
END_ACTION

ACTION _aN300_active:
// N300 — concurrent leg 1, first step. Everything a normal step does is available
// here; `Branch := 1` is what keeps this leg's issue latch, delay and message
// separate from the main line's, so both legs can command their own children in
// the same scan. This example commands nothing: the press has one work position,
// and inventing a second would change what the machine does. A real one goes here.
M_Step(StepNo := 300, StepName := 'project.step.pressParallelWork', Awaits := 0,
    AwaitingLabel := '', TimeClass := E_TimeClass.WORK, ExpectedTime := T#0S,
    Branch := 2);
_conRetVal[2] := E_StepResult.ADVANCE;   // leg 2's result; leg 1 uses _conRetVal[1]
END_ACTION

ACTION _aN310_active:
// N310 — concurrent leg 1 waits at the join. A parallel divergence joins only when
// EVERY leg has reached its last step, so each leg needs a terminal step to sit in
// while the others finish; this is that step for leg 1, and A250 is the main
// line's.
M_Step(StepNo := 310, StepName := 'project.step.pressAwaitParallelJoin', Awaits := 0,
    AwaitingLabel := '', TimeClass := E_TimeClass.WORK, ExpectedTime := T#0S,
    Branch := 2);
_conRetVal[2] := E_StepResult.ADVANCE;
END_ACTION

ACTION A000_Initialize:
// N000 step action. SFC step `A000_Initialize` calls this; its transition reads
// `_retVal = E_StepResult.ADVANCE`. Body is the ST chart's branch verbatim,
// without M_Advance - the chart runtime owns the transition.
M_Step(StepNo := 0, StepName := 'project.step.pressAutoInitialize',
    Awaits := 0, AwaitingLabel := '', TimeClass := E_TimeClass.WORK, ExpectedTime := T#0S, Branch := 0);
_outCmd.CycleCompleted := FALSE;
_retVal := E_StepResult.ADVANCE;
END_ACTION

ACTION A100_AwaitTwoHand:
// N100 step action. The §8.11.1 cycle-start marker; also the target of the
// N190 two-hand abort, which returns here with the same part still in place.
M_Step(StepNo := 100, StepName := 'project.step.pressAwaitTwoHand',
    Awaits := 0, AwaitingLabel := '', TimeClass := E_TimeClass.WAIT_OPERATOR, ExpectedTime := T#0S, Branch := 0);
_outCmd.CycleCompleted := FALSE;
_partReady := M_Await(Idx := 1, Label := 'project.condition.partPresent',
    Ok := _partPresentSensor.OutImm.Value AND _partPresentSensor.OutImm.Quality);
_airReady := M_Await(Idx := 2, Label := 'project.condition.airPressureOk',
    Ok := _airPressureMonitor.OutImm.PressureOk);
IF _stationCfg.RequireTwoHandStart THEN
    _startReady := M_Await(Idx := 3, Label := 'project.condition.twoHandStart', Ok := _startLatched);
ELSE
    _startReady := TRUE;
END_IF
IF M_StopPending() THEN
    M_StopNow();                       // stop accepted BETWEEN cycles: no phantom cycle
ELSIF _partReady AND _airReady AND _startReady THEN
    // §3.16.3 receive once per PHYSICAL part. The N180 two-hand abort returns
    // here with the same part still in the machine and nothing processed, so a
    // second M_PartReceived would open a duplicate record for one part.
    // M_PartStarted (N150) is deliberately NOT guarded: each pass is a genuine
    // processing attempt on that part.
    IF NOT _partInMachine THEN
        _traceAccepted := M_PartReceived();
        _partInMachine := TRUE;
    END_IF
    _retVal := E_StepResult.ADVANCE;
END_IF
END_ACTION

ACTION A110_RamUp:
// N110 step action. SFC step `A110_RamUp` calls this; its transition reads
// `_retVal = E_StepResult.ADVANCE`. Body is the ST chart's branch verbatim,
// without M_Advance - the chart runtime owns the transition.
M_Step(StepNo := 110, StepName := 'project.step.pressRamUp',
    Awaits := _pressRam, AwaitingLabel := 'PressRam.RETRACT', TimeClass := E_TimeClass.WORK, ExpectedTime := T#0S, Branch := 0);
IF M_TryIssue(Steppable := TRUE) THEN
    _pressRam.Abort := FALSE; _pressRam.Command := E_CylinderCommand.RETRACT; _pressRam.Execute := TRUE;
END_IF
IF _pressRam.Done THEN _pressRam.Execute := FALSE; _retVal := E_StepResult.ADVANCE; END_IF
END_ACTION

ACTION A130_DoorOpen:
// N130 step action. SFC step `A130_DoorOpen` calls this; its transition reads
// `_retVal = E_StepResult.ADVANCE`. Body is the ST chart's branch verbatim,
// without M_Advance - the chart runtime owns the transition.
M_Step(StepNo := 130, StepName := 'project.step.pressDoorOpen',
    Awaits := _door, AwaitingLabel := 'Door.RETRACT', TimeClass := E_TimeClass.WORK, ExpectedTime := T#0S, Branch := 0);
IF M_TryIssue(Steppable := TRUE) THEN
    _door.Abort := FALSE; _door.Command := E_CylinderCommand.RETRACT; _door.Execute := TRUE;
END_IF
IF _door.Done THEN _door.Execute := FALSE; _retVal := E_StepResult.ADVANCE; END_IF
END_ACTION

ACTION A150_SlideInside:
// N150 step action. SFC step `A150_SlideInside` calls this; its transition reads
// `_retVal = E_StepResult.ADVANCE`. Body is the ST chart's branch verbatim,
// without M_Advance - the chart runtime owns the transition.
M_Step(StepNo := 150, StepName := 'project.step.pressSlideInside',
    Awaits := _partSlide, AwaitingLabel := 'PartSlide.EXTEND', TimeClass := E_TimeClass.WORK, ExpectedTime := T#0S, Branch := 0);
IF M_TryIssue(Steppable := TRUE) THEN
    M_PartStarted();
    _partSlide.Abort := FALSE; _partSlide.Command := E_CylinderCommand.EXTEND; _partSlide.Execute := TRUE;
END_IF
IF _partSlide.Done THEN _partSlide.Execute := FALSE; _retVal := E_StepResult.ADVANCE; END_IF
END_ACTION

ACTION A170_TransferSettle:
// N170 step action. SFC step `A170_TransferSettle` calls this; its transition reads
// `_retVal = E_StepResult.ADVANCE`. Body is the ST chart's branch verbatim,
// without M_Advance - the chart runtime owns the transition.
M_Step(StepNo := 170, StepName := 'project.step.pressTransferSettle',
    Awaits := 0, AwaitingLabel := '', TimeClass := E_TimeClass.WORK, ExpectedTime := _parCfg.TransferSettleTime, Branch := 0);
_retVal := M_Delay(PT := _parCfg.TransferSettleTime);
END_ACTION

ACTION A180_DoorClose:
// N180 step action. Transition `_retVal = E_StepResult.ADVANCE` -> A200;
// the JUMP1 branch (`_retVal = E_StepResult.JUMP1`) -> A185.
//
// Releasing a two-hand button while the door is moving is an operator abort, not
// a fault: the door goes back up, the part slides out, and the cycle returns to
// the two-hand wait. Completion wins if the door finished in the same scan the
// button was released.
M_Step(StepNo := 180, StepName := 'project.step.pressDoorClose',
    Awaits := _door, AwaitingLabel := 'Door.EXTEND', TimeClass := E_TimeClass.WORK, ExpectedTime := T#0S, Branch := 0);
_twoHandHeldDuringClose := M_Await(Idx := 1,
    Label := 'project.condition.twoHandHeldDuringDoorClose',
    Ok := _twoHand.OutImm.SafeActive OR NOT _stationCfg.RequireTwoHandStart);
IF M_TryIssue(Steppable := TRUE) THEN
    _door.Abort := FALSE; _door.Command := E_CylinderCommand.EXTEND; _door.Execute := TRUE;
END_IF
IF _door.Done THEN
    _door.Execute := FALSE;
    _retVal := E_StepResult.ADVANCE;
ELSIF NOT _twoHandHeldDuringClose THEN
    _door.Execute := FALSE;             // §6.1 Execute-drop reset releases the close
    // §6.9(e) — a WARNING, not a fault: nothing stops, the JUMP1 branch below is
    // the recovery. Recorded because a cycle was abandoned with the part still in
    // the machine. Raised once per visit however many scans this action runs.
    _closeAbortWarned := M_RaiseWarning(
        Reason := PL_PressReasons.PRESS_TWO_HAND_RELEASED,
        DescriptionKey := 'project.warning.twoHandReleasedDuringDoorClose',
        Severity := E_Severity.LOW, Category := E_Category.PROCESS);
    _retVal := E_StepResult.JUMP1;      // released -> reopen and clear the part
END_IF
END_ACTION

ACTION A185_DoorReopen:
// N185 step action. Reached from A180 by JUMP1 when a two-hand button is
// released while the door closes. Advances to A190.
M_Step(StepNo := 185, StepName := 'project.step.pressDoorReopen',
    Awaits := _door, AwaitingLabel := 'Door.RETRACT', TimeClass := E_TimeClass.WORK, ExpectedTime := T#0S, Branch := 0);
IF M_TryIssue(Steppable := TRUE) THEN
    _door.Abort := FALSE; _door.Command := E_CylinderCommand.RETRACT; _door.Execute := TRUE;
END_IF
IF _door.Done THEN _door.Execute := FALSE; _retVal := E_StepResult.ADVANCE; END_IF
END_ACTION

ACTION A190_SlideOutsideAfterAbort:
// N190 step action. Slides the part out and drops the start latch, then its
// transition jumps back to A100, the two-hand wait. The start latch is dropped
// so the cycle cannot resume without a fresh two-hand press.
M_Step(StepNo := 190, StepName := 'project.step.pressSlideOutsideAfterAbort',
    Awaits := _partSlide, AwaitingLabel := 'PartSlide.RETRACT', TimeClass := E_TimeClass.WORK, ExpectedTime := T#0S, Branch := 0);
IF M_TryIssue(Steppable := TRUE) THEN
    _partSlide.Abort := FALSE; _partSlide.Command := E_CylinderCommand.RETRACT; _partSlide.Execute := TRUE;
END_IF
IF _partSlide.Done THEN
    _partSlide.Execute := FALSE;
    _startLatched := FALSE;
    _retVal := E_StepResult.ADVANCE;
END_IF
END_ACTION

ACTION A200_RamDown:
// N200 step action. Transition `_retVal = E_StepResult.ADVANCE` -> A220;
// the JUMP1 branch (`_retVal = E_StepResult.JUMP1`) -> A210.
// the ram to the §6.9 auto-rollup: an awaited child fault is adopted by the
// Unit (ERROR, _step := 0) before _M_Dispatch runs, and the chain would stop
// before it could ask the operator anything. The wait is still named (§6.9(b))
// and the cylinder still raises its own CYL_NOT_EXTENDED alarm.
M_Step(StepNo := 200, StepName := 'project.step.pressRamDown',
    Awaits := 0, AwaitingLabel := '', TimeClass := E_TimeClass.WORK, ExpectedTime := T#0S,
    Branch := 1);
_ramReached := M_Await(Idx := 1, Label := 'project.condition.pressRamExtended',
    Ok := _pressRam.Done);
IF M_TryIssue(Steppable := TRUE) THEN
    _pressRam.Abort := FALSE; _pressRam.Command := E_CylinderCommand.EXTEND; _pressRam.Execute := TRUE;
END_IF
IF _pressRam.Done THEN
    _pressRam.Execute := FALSE;
    _conRetVal[1] := E_StepResult.ADVANCE;
ELSIF _pressRam.Error THEN
    // §6.9(e) — publish the ram's own first-out on the Unit and on this row of the
    // §3.13 chart without adopting it: the confirmation + scrap below IS the
    // handling, so a fault here would replace a designed recovery.
    _ramFailureReported := M_ReportFromChild(Source := _pressRam);
    _pressRam.Execute := FALSE;         // §6.1 Execute-drop reset returns the ram to READY
    _conRetVal[1] := E_StepResult.JUMP1;      // did not reach -> operator confirmation
END_IF
END_ACTION

ACTION A210_ConfirmPressFailure:
// N210 step action. Reached from A200 by JUMP1; advances to A215.
// scrapped. A scrap is deliberate, so there is no timeout default (§6.11).
M_Step(StepNo := 210, StepName := 'project.step.pressNotReachedConfirm',
    Awaits := 0, AwaitingLabel := '', TimeClass := E_TimeClass.WAIT_OPERATOR, ExpectedTime := T#0S,
    Branch := 1);
_decisionRequest.Prompt := 'project.decision.pressNotReached';
_decisionRequest.Options[1] := 'project.decision.confirmScrapAndReturn';
_decisionRequest.Default := 0;
_decisionRequest.Timeout := T#0S;
M_AskDecision(Req := _decisionRequest);
_answer := M_TakeDecision();
IF _answer = 1 THEN
    _conRetVal[1] := E_StepResult.ADVANCE;
ELSE
    _failureConfirmed := M_Await(Idx := 1,
        Label := 'project.condition.pressFailureConfirmation', Ok := FALSE);
END_IF
END_ACTION

ACTION A215_ScrapPart:
// N215 step action. Sets the part NOK and releases it, then rejoins A240.
M_Step(StepNo := 215, StepName := 'project.step.pressScrapPart',
    Awaits := 0, AwaitingLabel := '', TimeClass := E_TimeClass.WORK, ExpectedTime := T#0S,
    Branch := 1);
_partProcessed := M_PartProcessed(Verdict := E_Verdict.NOK,
    Reason := PL_ModuleReasons.CYL_NOT_EXTENDED);
_partDispositioned := TRUE;             // N999 must not also count it good
_partInMachine := FALSE;                // dispositioned: the next one is a new part
_outCmd.CycleCompleted := FALSE;
_conRetVal[1] := E_StepResult.ADVANCE;
END_ACTION

ACTION A220_PressDwell:
// N220 step action. SFC step `A220_PressDwell` calls this; its transition reads
// `_retVal = E_StepResult.ADVANCE`. Body is the ST chart's branch verbatim,
// without M_Advance - the chart runtime owns the transition.
M_Step(StepNo := 220, StepName := 'project.step.pressDwell',
    Awaits := 0, AwaitingLabel := '', TimeClass := E_TimeClass.WORK, ExpectedTime := _parCfg.PressSettleTime,
    Branch := 1);
// Releasing the button mid-dwell is the designed way to stop pressing, so it
// is a named wait (§6.9(b)), not a fault: the ram's outputs come off, the
// dwell timer freezes where it is because M_Delay is not called, and pressing
// again restores the force and finishes the remaining dwell. Faulting here
// charged an unrecoverable downtime event for normal operator behaviour.
_dwellTwoHandHeld := M_Await(Idx := 1, Label := 'project.condition.twoHandHeldDuringPress',
    Ok := _twoHand.OutImm.SafeActive OR NOT _stationCfg.RequireTwoHandStart);
IF NOT _dwellTwoHandHeld THEN
    _pressRam.WithdrawOutputs();
ELSE
    // The press force is the valve latched by the EXTEND that step 200 already
    // completed, so after a withdraw only this call re-energizes it — and the
    // ram re-checks its own extend permit before it does (§7.2).
    _pressRam.RestoreOutputs();
    _conRetVal[1] := M_Delay(PT := _parCfg.PressSettleTime);
END_IF
END_ACTION

ACTION A230_RecordResult:
// N230 step action. SFC step `A230_RecordResult` calls this; its transition reads
// `_retVal = E_StepResult.ADVANCE`. Body is the ST chart's branch verbatim,
// without M_Advance - the chart runtime owns the transition.
M_Step(StepNo := 230, StepName := 'project.step.pressRecordResult',
    Awaits := 0, AwaitingLabel := '', TimeClass := E_TimeClass.WORK, ExpectedTime := T#0S,
    Branch := 1);
_recordAccepted := M_PartRecord(RecordName := 'PressDwell',
    Value := DINT_TO_LREAL(TIME_TO_DINT(_parCfg.PressSettleTime)),
    Minimum := 0, Maximum := 30000,
    Target := DINT_TO_LREAL(TIME_TO_DINT(_parCfg.PressSettleTime)), EngUnit := 'ms');
_conRetVal[1] := E_StepResult.ADVANCE;
END_ACTION

ACTION A240_ReturnToLoadPosition:
// N240 step action, on concurrent leg 1. Its transition reads
// `_conRetVal[1] = E_StepResult.ADVANCE`. Body is the ST chart's branch verbatim,
// without M_Advance - the chart runtime owns the transition.
//
// The sub-chain needs no leg argument: M_RunSub inherits the leg of the step that
// runs it (§6.12), so the load-position steps publish as leg 1 too.
_conRetVal[1] := M_RunSub(Chain := _loadPosition, BaseStepNo := 240);
END_ACTION

ACTION A999_CycleComplete:
// N999 step action. Transition `_retVal = E_StepResult.ADVANCE` loops to A100.
M_Step(StepNo := 999, StepName := 'project.step.pressAutoComplete',
    Awaits := 0, AwaitingLabel := '', TimeClass := E_TimeClass.WORK, ExpectedTime := T#0S, Branch := 0);
_outCmd.CycleCompleted := TRUE;
IF _partDispositioned THEN
    _partDispositioned := FALSE;       // N260 already set the NOK verdict
ELSE
    _partProcessed := M_PartProcessed(Verdict := E_Verdict.OK, Reason := E_Reason.NONE);
    IF NOT _partProcessed THEN
        M_CountGood();                 // §3.9: no carrier configured — count directly
    END_IF
END_IF
_partInMachine := FALSE;               // processed: the next one is a new part
_startLatched := FALSE;
IF M_EndOfCycle() THEN
    _retVal := E_StepResult.ADVANCE;   // stop NOT requested: loop to N100
END_IF
END_ACTION

// §6.8 - the chain's own state on a restart (the base resets the flow state).
METHOD PROTECTED OnChainReset
// A chart restart abandons whatever the cycle was holding: the part record is
// closed by N215/N999, never by a restart, so both trackers start clean.
_partDispositioned := FALSE;
_partInMachine := FALSE;
END_METHOD

METHOD Setup : BOOL
VAR_INPUT
    Host : I_SequenceHost;
END_VAR
VAR_IN_OUT
    PressRam : FB_CylinderCM;
    Door : FB_CylinderCM;
    PartSlide : FB_CylinderCM;
    TwoHand : FB_TwoHandStartCM;
    PartPresentSensor : FB_DigitalInputCM;
    AirPressureMonitor : FB_AirPressureMonitorCM;
    ParCfg : ST_PneumaticPressParCfg;
    StationCfg : ST_PneumaticPressStationCfg;
    OutCmd : ST_PneumaticPressOutCmd;
    StartLatched : BOOL;
END_VAR
_pressRam REF= PressRam;
_door REF= Door;
_partSlide REF= PartSlide;
_twoHand REF= TwoHand;
_partPresentSensor REF= PartPresentSensor;
_airPressureMonitor REF= AirPressureMonitor;
_parCfg REF= ParCfg;
_stationCfg REF= StationCfg;
_outCmd REF= OutCmd;
_startLatched REF= StartLatched;
Setup := M_Attach(Host := Host) AND __ISVALIDREF(_pressRam) AND __ISVALIDREF(_door)
    AND __ISVALIDREF(_partSlide) AND __ISVALIDREF(_twoHand)
    AND __ISVALIDREF(_partPresentSensor) AND __ISVALIDREF(_airPressureMonitor)
    AND __ISVALIDREF(_parCfg) AND __ISVALIDREF(_outCmd) AND __ISVALIDREF(_startLatched)
    AND _loadPosition.Setup(Host := Host, PressRam := PressRam, Door := Door, PartSlide := PartSlide);
END_METHOD

END_FUNCTION_BLOCK

// ---- 01_PneumaticPress/Sequences/FB_LD_PressDemoAuto.TcPOU
FUNCTION_BLOCK FB_LD_PressDemoAuto EXTENDS FB_SequenceBase
VAR
    _partReady, _airReady, _startReady, _stop, _doStep, _processed, _endCycle, _dummy : BOOL;
    _dwellTwoHandHeld : BOOL;          // N220 named wait: two-hand held through the dwell
    _decisionRequest : ST_DecisionRequest;   // §6.11 not-reached confirmation
    _answer : INT;
    _ramReached, _failureConfirmed : BOOL;   // N200/N210 named waits
    _twoHandHeldDuringClose : BOOL;          // N180 named wait
    _closeAbortWarned : BOOL;                // N180 §6.9(e) message result
    _ramFailureReported : BOOL;              // N200 §6.9(e) message result
    _partInMachine : BOOL;                   // §3.16.3 the part is already received
    _partDispositioned : BOOL;               // N260 already set the verdict
    _traceAccepted, _recordAccepted, _partProcessed : BOOL;
    {attribute 'OPC.UA.DA' := '0'}
    _pressRam : REFERENCE TO FB_CylinderCM;
    {attribute 'OPC.UA.DA' := '0'}
    _door : REFERENCE TO FB_CylinderCM;
    {attribute 'OPC.UA.DA' := '0'}
    _partSlide : REFERENCE TO FB_CylinderCM;
    {attribute 'OPC.UA.DA' := '0'}
    _twoHand : REFERENCE TO FB_TwoHandStartCM;
    {attribute 'OPC.UA.DA' := '0'}
    _partPresentSensor : REFERENCE TO FB_DigitalInputCM;
    {attribute 'OPC.UA.DA' := '0'}
    _airPressureMonitor : REFERENCE TO FB_AirPressureMonitorCM;
    {attribute 'OPC.UA.DA' := '0'}
    _parCfg : REFERENCE TO ST_PneumaticPressParCfg;
    // §3.8a - the cell's own policy, referenced like _parCfg.
    {attribute 'OPC.UA.DA' := '0'}
    _stationCfg : REFERENCE TO ST_PneumaticPressStationCfg;
    {attribute 'OPC.UA.DA' := '0'}
    _outCmd : REFERENCE TO ST_PneumaticPressOutCmd;
    {attribute 'OPC.UA.DA' := '0'}
    _startLatched : REFERENCE TO BOOL;
    {attribute 'OPC.UA.DA' := '0'}
    _loadPosition : FB_PressDemoLoadPosition;
END_VAR
VAR // added by the converter: edge detectors and wires of the graphical bodies
    _w1, _w2, _w3, _w4, _w5, _w6, _w7, _w8, _w9, _w10, _w11, _w12, _w13, _w14, _w15, _w16, _w17, _w18, _w19, _w20, _w21, _w22, _w23, _w24, _w25, _w26, _w27, _w28, _w29, _w30 : BOOL;
END_VAR

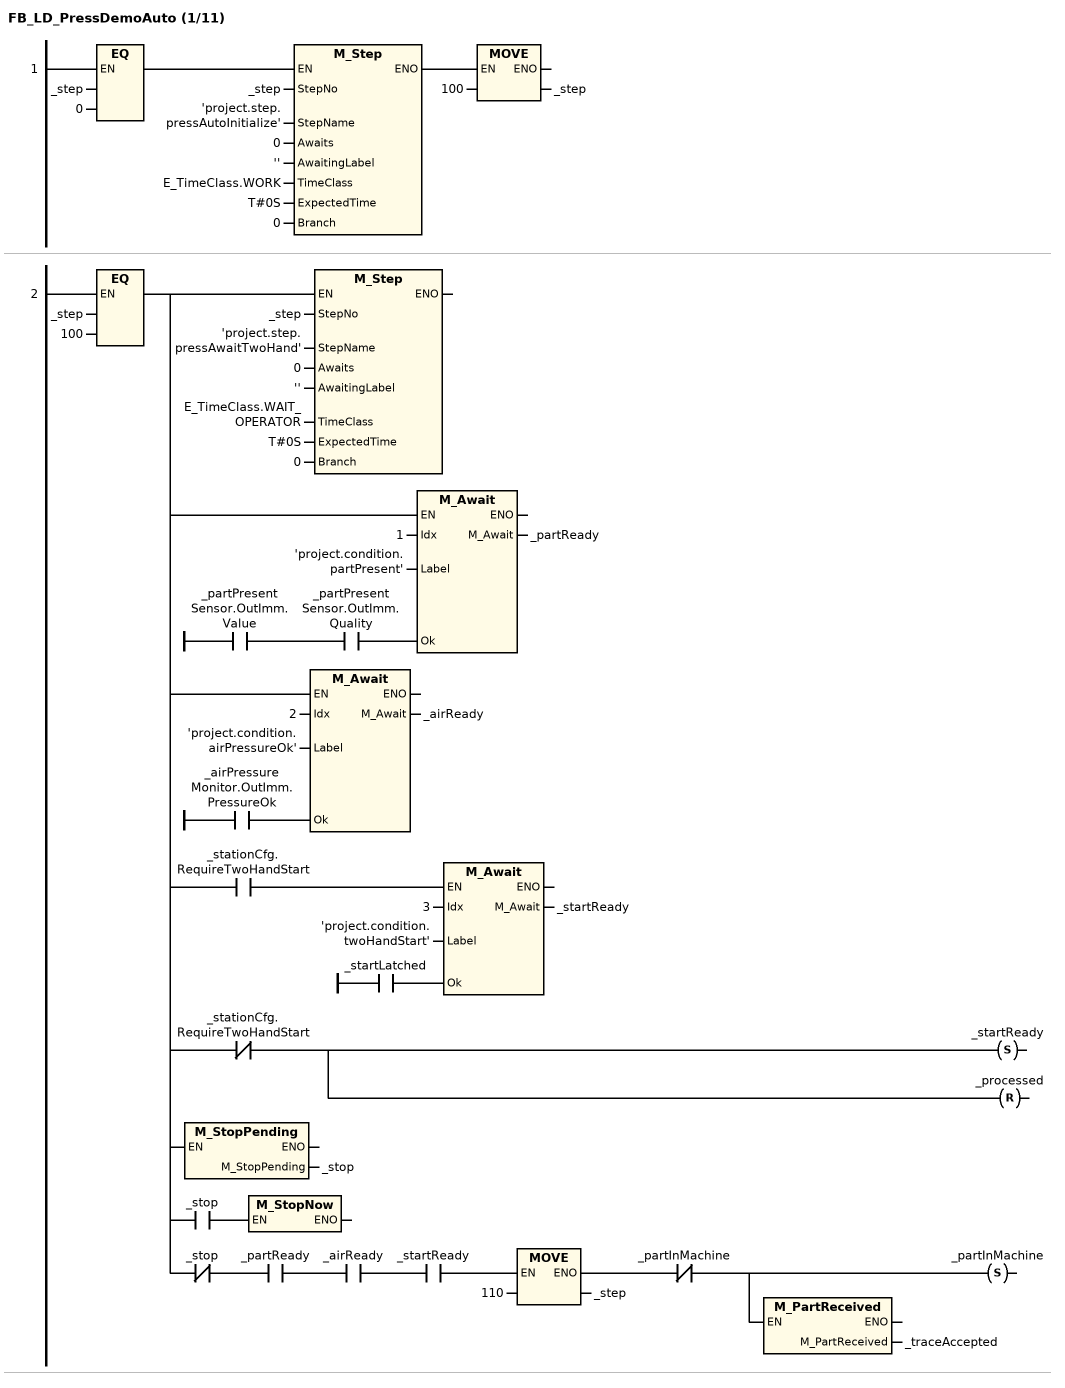
// NETWORK 1
_w1 := _step = 0;
IF _w1 THEN
    M_Step(StepNo := _step, StepName := 'project.step.pressAutoInitialize', Awaits := 0, AwaitingLabel := '', TimeClass := E_TimeClass.WORK, ExpectedTime := T#0S, Branch := 0);
END_IF
IF _w1 THEN _step := 100; END_IF

// NETWORK 2
_w2 := _step = 100;
IF _w2 THEN
    M_Step(StepNo := _step, StepName := 'project.step.pressAwaitTwoHand', Awaits := 0, AwaitingLabel := '', TimeClass := E_TimeClass.WAIT_OPERATOR, ExpectedTime := T#0S, Branch := 0);
END_IF
IF _w2 THEN
    _partReady := M_Await(Idx := 1, Label := 'project.condition.partPresent', Ok := _partPresentSensor.OutImm.Value AND _partPresentSensor.OutImm.Quality);
END_IF
IF _w2 THEN
    _airReady := M_Await(Idx := 2, Label := 'project.condition.airPressureOk', Ok := _airPressureMonitor.OutImm.PressureOk);
END_IF
IF _w2 AND _stationCfg.RequireTwoHandStart THEN
    _startReady := M_Await(Idx := 3, Label := 'project.condition.twoHandStart', Ok := _startLatched);
END_IF
_w3 := _w2 AND NOT _stationCfg.RequireTwoHandStart;
_startReady S= _w3;
_processed R= _w3;
IF _w2 THEN _stop := M_StopPending(); END_IF
IF _w2 AND _stop THEN M_StopNow(); END_IF
IF _w2 AND NOT _stop AND _partReady AND _airReady AND _startReady THEN _step := 110; END_IF
_w4 := (_w2 AND NOT _stop AND _partReady AND _airReady AND _startReady) AND NOT _partInMachine;
_partInMachine S= _w4;
IF _w4 THEN _traceAccepted := M_PartReceived(); END_IF

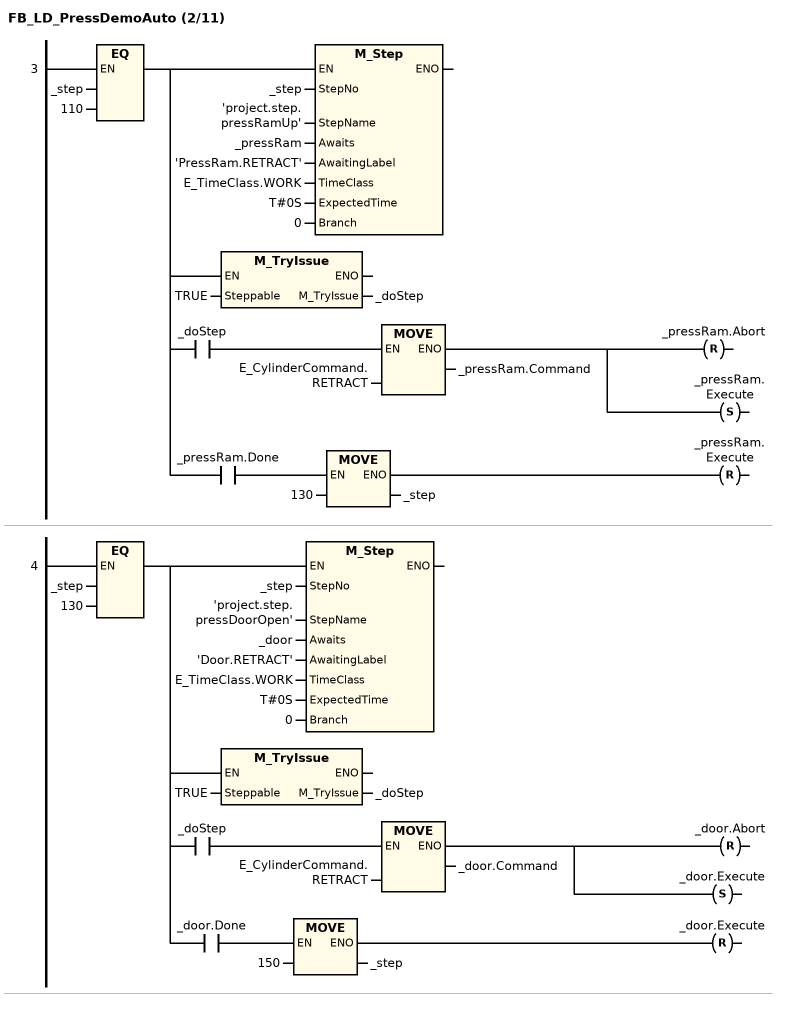
// NETWORK 3
_w5 := _step = 110;
IF _w5 THEN
    M_Step(StepNo := _step, StepName := 'project.step.pressRamUp', Awaits := _pressRam, AwaitingLabel := 'PressRam.RETRACT', TimeClass := E_TimeClass.WORK, ExpectedTime := T#0S, Branch := 0);
END_IF
IF _w5 THEN _doStep := M_TryIssue(Steppable := TRUE); END_IF
IF _w5 AND _doStep THEN _pressRam.Command := E_CylinderCommand.RETRACT; END_IF
_w6 := _w5 AND _doStep;
_pressRam.Abort R= _w6;
_pressRam.Execute S= _w6;
IF _w5 AND _pressRam.Done THEN _step := 130; END_IF
_pressRam.Execute R= _w5 AND _pressRam.Done;

// NETWORK 4
_w7 := _step = 130;
IF _w7 THEN
    M_Step(StepNo := _step, StepName := 'project.step.pressDoorOpen', Awaits := _door, AwaitingLabel := 'Door.RETRACT', TimeClass := E_TimeClass.WORK, ExpectedTime := T#0S, Branch := 0);
END_IF
IF _w7 THEN _doStep := M_TryIssue(Steppable := TRUE); END_IF
IF _w7 AND _doStep THEN _door.Command := E_CylinderCommand.RETRACT; END_IF
_w8 := _w7 AND _doStep;
_door.Abort R= _w8;
_door.Execute S= _w8;
IF _w7 AND _door.Done THEN _step := 150; END_IF
_door.Execute R= _w7 AND _door.Done;

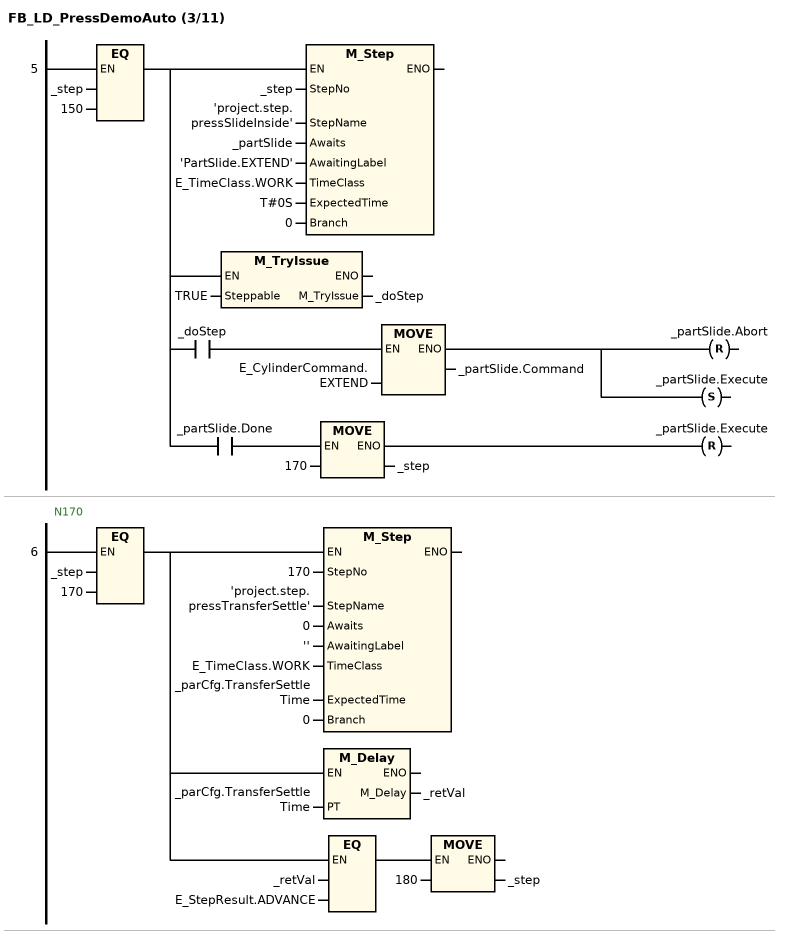
// NETWORK 5
_w9 := _step = 150;
IF _w9 THEN
    M_Step(StepNo := _step, StepName := 'project.step.pressSlideInside', Awaits := _partSlide, AwaitingLabel := 'PartSlide.EXTEND', TimeClass := E_TimeClass.WORK, ExpectedTime := T#0S, Branch := 0);
END_IF
IF _w9 THEN _doStep := M_TryIssue(Steppable := TRUE); END_IF
IF _w9 AND _doStep THEN _partSlide.Command := E_CylinderCommand.EXTEND; END_IF
_w10 := _w9 AND _doStep;
_partSlide.Abort R= _w10;
_partSlide.Execute S= _w10;
IF _w9 AND _partSlide.Done THEN _step := 170; END_IF
_partSlide.Execute R= _w9 AND _partSlide.Done;

// NETWORK 6
// N170
_w11 := _step = 170;
IF _w11 THEN
    M_Step(StepNo := 170, StepName := 'project.step.pressTransferSettle', Awaits := 0, AwaitingLabel := '', TimeClass := E_TimeClass.WORK, ExpectedTime := _parCfg.TransferSettleTime, Branch := 0);
END_IF
IF _w11 THEN _retVal := M_Delay(PT := _parCfg.TransferSettleTime); END_IF
IF _w11 AND _retVal = E_StepResult.ADVANCE THEN _step := 180; END_IF

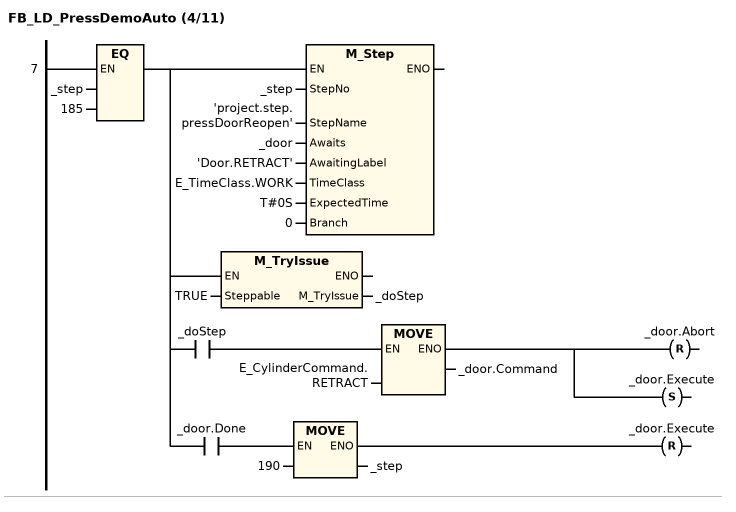
// NETWORK 7
_w12 := _step = 185;
IF _w12 THEN
    M_Step(StepNo := _step, StepName := 'project.step.pressDoorReopen', Awaits := _door, AwaitingLabel := 'Door.RETRACT', TimeClass := E_TimeClass.WORK, ExpectedTime := T#0S, Branch := 0);
END_IF
IF _w12 THEN _doStep := M_TryIssue(Steppable := TRUE); END_IF
IF _w12 AND _doStep THEN _door.Command := E_CylinderCommand.RETRACT; END_IF
_w13 := _w12 AND _doStep;
_door.Abort R= _w13;
_door.Execute S= _w13;
IF _w12 AND _door.Done THEN _step := 190; END_IF
_door.Execute R= _w12 AND _door.Done;

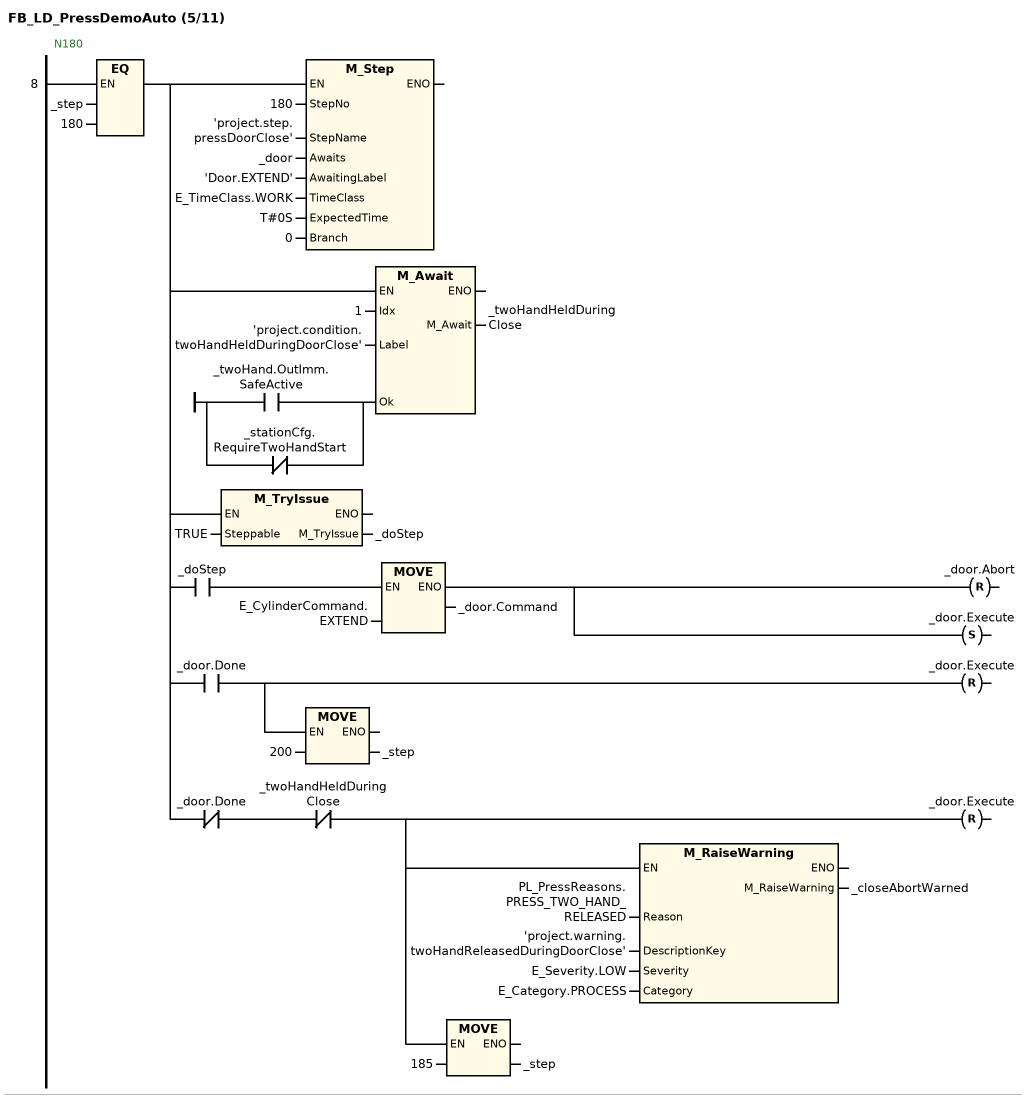
// NETWORK 8
// N180
_w14 := _step = 180;
IF _w14 THEN
    M_Step(StepNo := 180, StepName := 'project.step.pressDoorClose', Awaits := _door, AwaitingLabel := 'Door.EXTEND', TimeClass := E_TimeClass.WORK, ExpectedTime := T#0S, Branch := 0);
END_IF
IF _w14 THEN
    _twoHandHeldDuringClose := M_Await(Idx := 1, Label := 'project.condition.twoHandHeldDuringDoorClose', Ok := _twoHand.OutImm.SafeActive OR NOT _stationCfg.RequireTwoHandStart);
END_IF
IF _w14 THEN _doStep := M_TryIssue(Steppable := TRUE); END_IF
IF _w14 AND _doStep THEN _door.Command := E_CylinderCommand.EXTEND; END_IF
_w15 := _w14 AND _doStep;
_door.Abort R= _w15;
_door.Execute S= _w15;
_w16 := _w14 AND _door.Done;
_door.Execute R= _w16;
IF _w16 THEN _step := 200; END_IF
_w17 := _w14 AND NOT _door.Done AND NOT _twoHandHeldDuringClose;
_door.Execute R= _w17;
IF _w17 THEN
    _closeAbortWarned := M_RaiseWarning(Reason := PL_PressReasons.PRESS_TWO_HAND_RELEASED, DescriptionKey := 'project.warning.twoHandReleasedDuringDoorClose', Severity := E_Severity.LOW, Category := E_Category.PROCESS);
END_IF
IF _w17 THEN _step := 185; END_IF

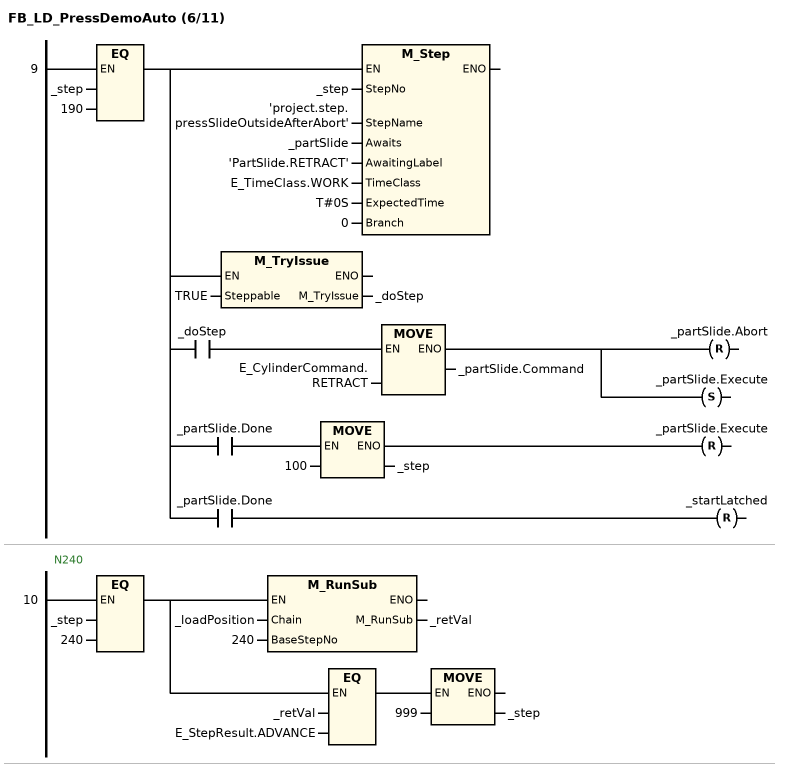
// NETWORK 9
_w18 := _step = 190;
IF _w18 THEN
    M_Step(StepNo := _step, StepName := 'project.step.pressSlideOutsideAfterAbort', Awaits := _partSlide, AwaitingLabel := 'PartSlide.RETRACT', TimeClass := E_TimeClass.WORK, ExpectedTime := T#0S, Branch := 0);
END_IF
IF _w18 THEN _doStep := M_TryIssue(Steppable := TRUE); END_IF
IF _w18 AND _doStep THEN _partSlide.Command := E_CylinderCommand.RETRACT; END_IF
_w19 := _w18 AND _doStep;
_partSlide.Abort R= _w19;
_partSlide.Execute S= _w19;
IF _w18 AND _partSlide.Done THEN _step := 100; END_IF
_partSlide.Execute R= _w18 AND _partSlide.Done;
_startLatched R= _w18 AND _partSlide.Done;

// NETWORK 10
// N240
_w20 := _step = 240;
IF _w20 THEN _retVal := M_RunSub(Chain := _loadPosition, BaseStepNo := 240); END_IF
IF _w20 AND _retVal = E_StepResult.ADVANCE THEN _step := 999; END_IF

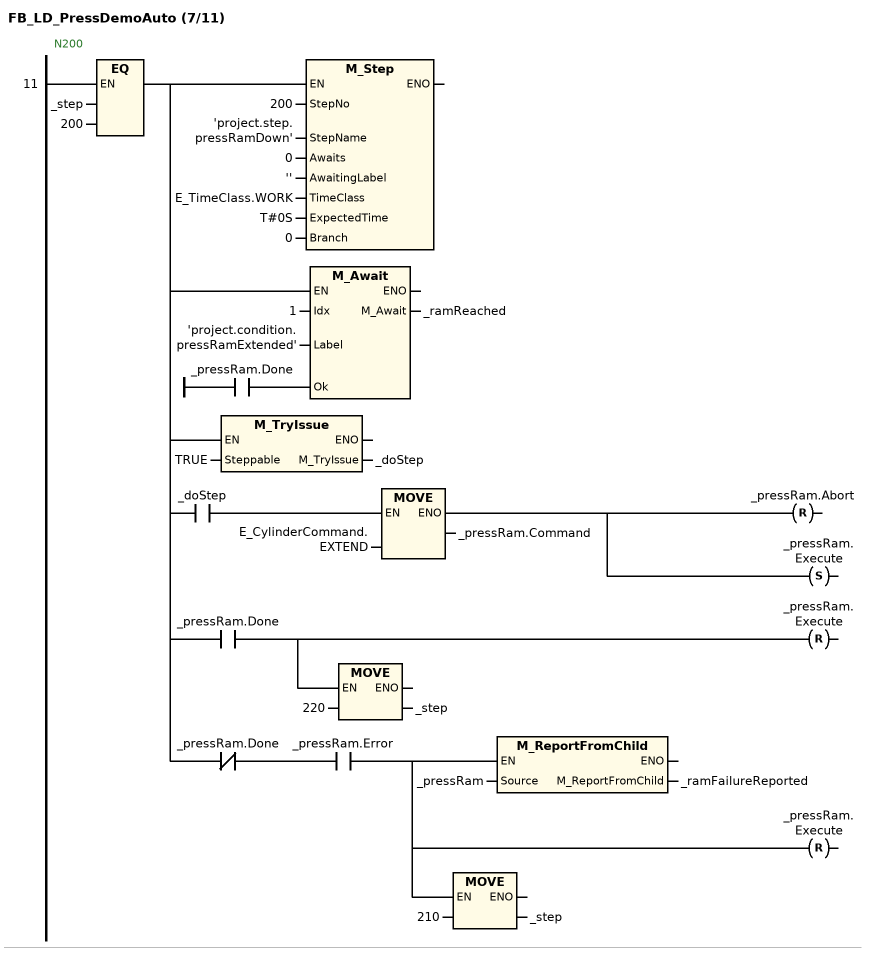
// NETWORK 11
// N200
_w21 := _step = 200;
IF _w21 THEN
    M_Step(StepNo := 200, StepName := 'project.step.pressRamDown', Awaits := 0, AwaitingLabel := '', TimeClass := E_TimeClass.WORK, ExpectedTime := T#0S, Branch := 0);
END_IF
IF _w21 THEN
    _ramReached := M_Await(Idx := 1, Label := 'project.condition.pressRamExtended', Ok := _pressRam.Done);
END_IF
IF _w21 THEN _doStep := M_TryIssue(Steppable := TRUE); END_IF
IF _w21 AND _doStep THEN _pressRam.Command := E_CylinderCommand.EXTEND; END_IF
_w22 := _w21 AND _doStep;
_pressRam.Abort R= _w22;
_pressRam.Execute S= _w22;
_w23 := _w21 AND _pressRam.Done;
_pressRam.Execute R= _w23;
IF _w23 THEN _step := 220; END_IF
_w24 := _w21 AND NOT _pressRam.Done AND _pressRam.Error;
IF _w24 THEN _ramFailureReported := M_ReportFromChild(Source := _pressRam); END_IF
_pressRam.Execute R= _w24;
IF _w24 THEN _step := 210; END_IF

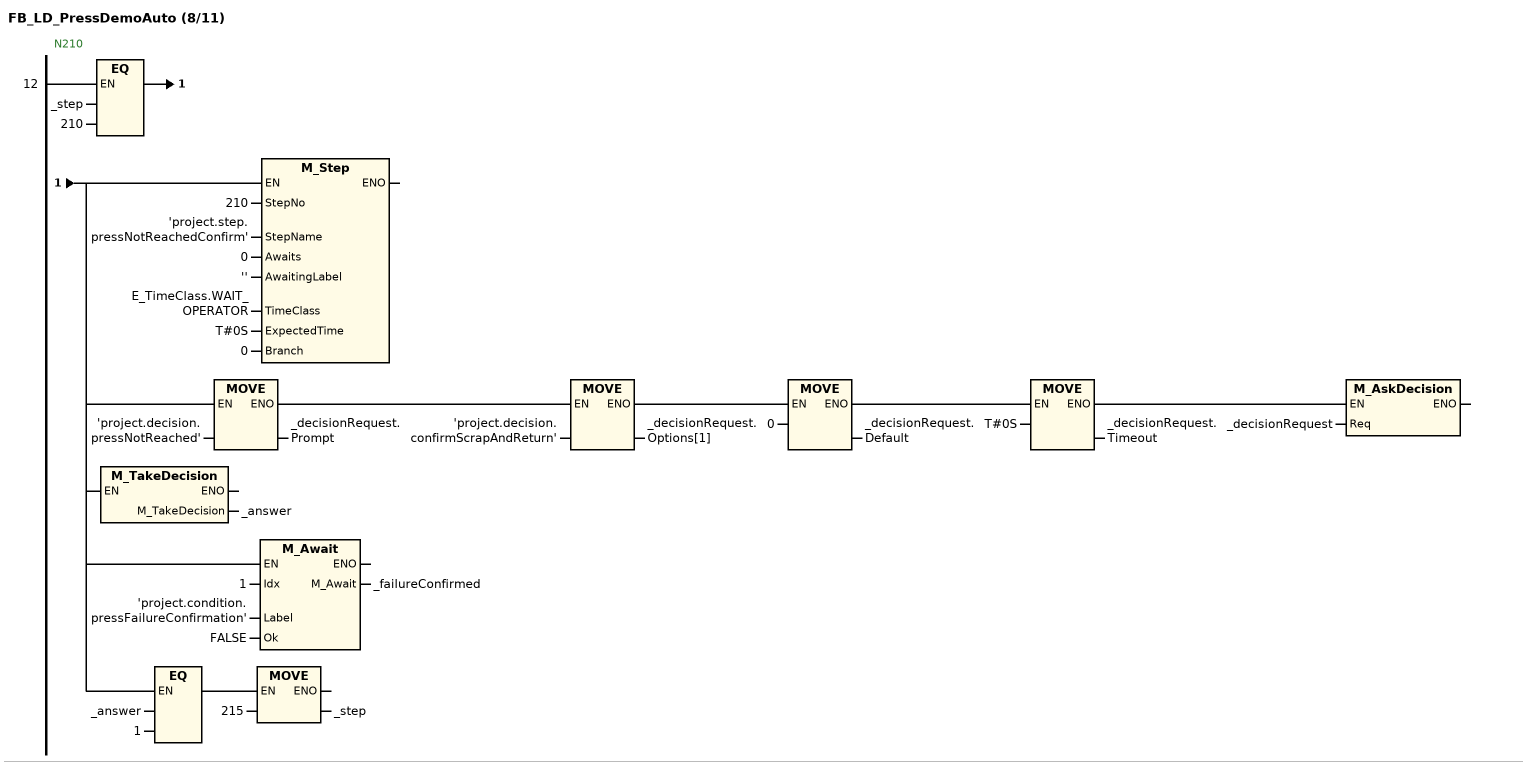
// NETWORK 12
// N210
_w25 := _step = 210;
IF _w25 THEN
    M_Step(StepNo := 210, StepName := 'project.step.pressNotReachedConfirm', Awaits := 0, AwaitingLabel := '', TimeClass := E_TimeClass.WAIT_OPERATOR, ExpectedTime := T#0S, Branch := 0);
END_IF
IF _w25 THEN _decisionRequest.Prompt := 'project.decision.pressNotReached'; END_IF
IF _w25 THEN _decisionRequest.Options[1] := 'project.decision.confirmScrapAndReturn'; END_IF
IF _w25 THEN _decisionRequest.Default := 0; END_IF
IF _w25 THEN _decisionRequest.Timeout := T#0S; END_IF
IF _w25 THEN M_AskDecision(Req := _decisionRequest); END_IF
IF _w25 THEN _answer := M_TakeDecision(); END_IF
IF _w25 THEN
    _failureConfirmed := M_Await(Idx := 1, Label := 'project.condition.pressFailureConfirmation', Ok := FALSE);
END_IF
IF _w25 AND _answer = 1 THEN _step := 215; END_IF

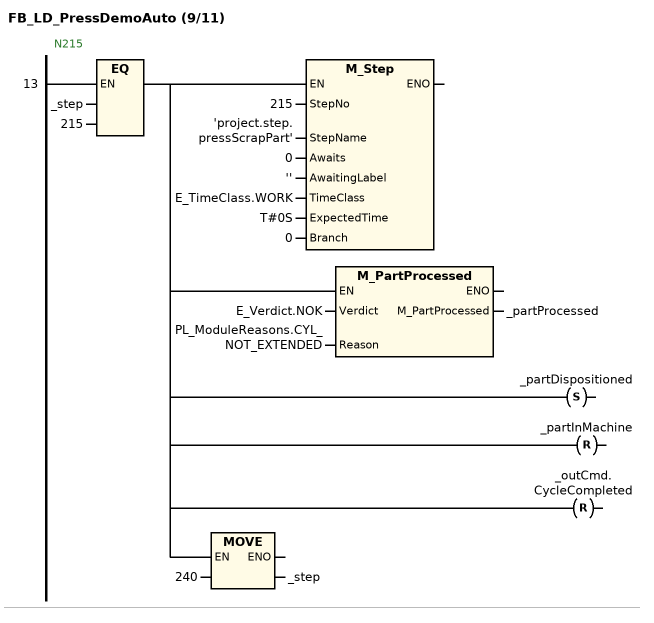
// NETWORK 13
// N215
_w26 := _step = 215;
IF _w26 THEN
    M_Step(StepNo := 215, StepName := 'project.step.pressScrapPart', Awaits := 0, AwaitingLabel := '', TimeClass := E_TimeClass.WORK, ExpectedTime := T#0S, Branch := 0);
END_IF
IF _w26 THEN
    _partProcessed := M_PartProcessed(Verdict := E_Verdict.NOK, Reason := PL_ModuleReasons.CYL_NOT_EXTENDED);
END_IF
_partDispositioned S= _w26;
_partInMachine R= _w26;
_outCmd.CycleCompleted R= _w26;
IF _w26 THEN _step := 240; END_IF

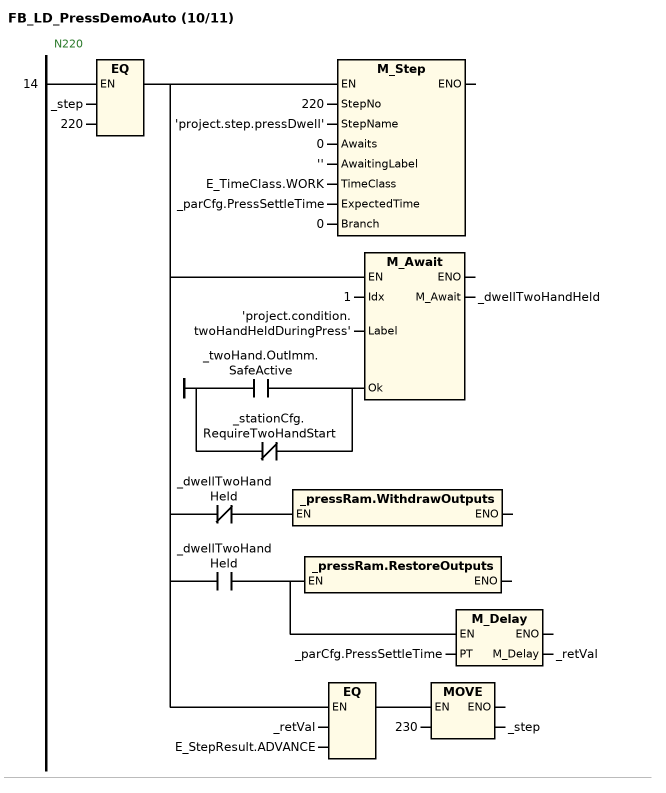
// NETWORK 14
// N220
_w27 := _step = 220;
IF _w27 THEN
    M_Step(StepNo := 220, StepName := 'project.step.pressDwell', Awaits := 0, AwaitingLabel := '', TimeClass := E_TimeClass.WORK, ExpectedTime := _parCfg.PressSettleTime, Branch := 0);
END_IF
IF _w27 THEN
    _dwellTwoHandHeld := M_Await(Idx := 1, Label := 'project.condition.twoHandHeldDuringPress', Ok := _twoHand.OutImm.SafeActive OR NOT _stationCfg.RequireTwoHandStart);
END_IF
IF _w27 AND NOT _dwellTwoHandHeld THEN _pressRam.WithdrawOutputs(); END_IF
_w28 := _w27 AND _dwellTwoHandHeld;
IF _w28 THEN _pressRam.RestoreOutputs(); END_IF
IF _w28 THEN _retVal := M_Delay(PT := _parCfg.PressSettleTime); END_IF
IF _w27 AND _retVal = E_StepResult.ADVANCE THEN _step := 230; END_IF

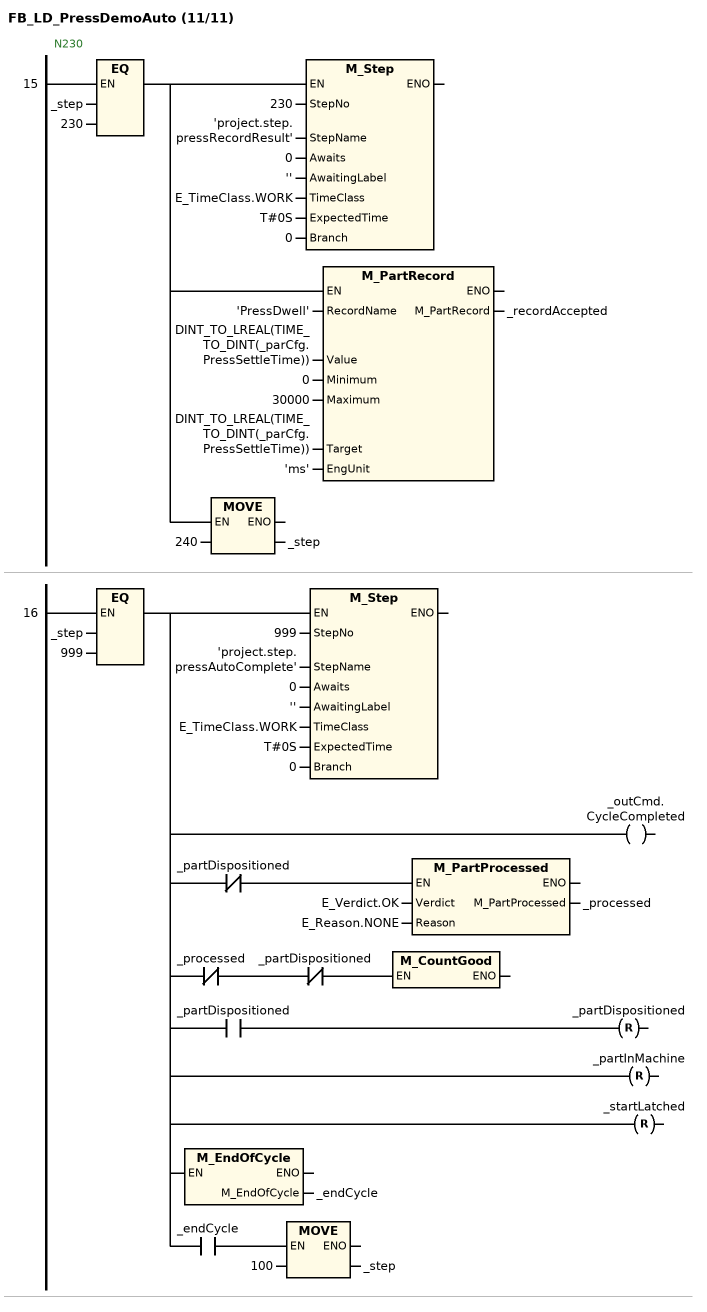
// NETWORK 15
// N230
_w29 := _step = 230;
IF _w29 THEN
    M_Step(StepNo := 230, StepName := 'project.step.pressRecordResult', Awaits := 0, AwaitingLabel := '', TimeClass := E_TimeClass.WORK, ExpectedTime := T#0S, Branch := 0);
END_IF
IF _w29 THEN
    _recordAccepted := M_PartRecord(RecordName := 'PressDwell', Value := DINT_TO_LREAL(TIME_TO_DINT(_parCfg.PressSettleTime)), Minimum := 0, Maximum := 30000, Target := DINT_TO_LREAL(TIME_TO_DINT(_parCfg.PressSettleTime)), EngUnit := 'ms');
END_IF
IF _w29 THEN _step := 240; END_IF

// NETWORK 16
_w30 := _step = 999;
IF _w30 THEN
    M_Step(StepNo := 999, StepName := 'project.step.pressAutoComplete', Awaits := 0, AwaitingLabel := '', TimeClass := E_TimeClass.WORK, ExpectedTime := T#0S, Branch := 0);
END_IF
_outCmd.CycleCompleted := _w30;
IF _w30 AND NOT _partDispositioned THEN
    _processed := M_PartProcessed(Verdict := E_Verdict.OK, Reason := E_Reason.NONE);
END_IF
IF _w30 AND NOT _processed AND NOT _partDispositioned THEN M_CountGood(); END_IF
_partDispositioned R= _w30 AND _partDispositioned;
_partInMachine R= _w30;
_startLatched R= _w30;
IF _w30 THEN _endCycle := M_EndOfCycle(); END_IF
IF _w30 AND _endCycle THEN _step := 100; END_IF

// Identical signature to the ST and SFC renditions of this chain, so the Unit can
// bind whichever one AUTO_SEQUENCE_LANGUAGE selects without any other difference.
METHOD Setup : BOOL
VAR_INPUT
    Host : I_SequenceHost;
END_VAR
VAR_IN_OUT
    PressRam : FB_CylinderCM;
    Door : FB_CylinderCM;
    PartSlide : FB_CylinderCM;
    TwoHand : FB_TwoHandStartCM;
    PartPresentSensor : FB_DigitalInputCM;
    AirPressureMonitor : FB_AirPressureMonitorCM;
    ParCfg : ST_PneumaticPressParCfg;
    StationCfg : ST_PneumaticPressStationCfg;
    OutCmd : ST_PneumaticPressOutCmd;
    StartLatched : BOOL;
END_VAR
_pressRam REF= PressRam;
_door REF= Door;
_partSlide REF= PartSlide;
_twoHand REF= TwoHand;
_partPresentSensor REF= PartPresentSensor;
_airPressureMonitor REF= AirPressureMonitor;
_parCfg REF= ParCfg;
_stationCfg REF= StationCfg;
_outCmd REF= OutCmd;
_startLatched REF= StartLatched;
Setup := M_Attach(Host := Host) AND __ISVALIDREF(_pressRam) AND __ISVALIDREF(_door)
    AND __ISVALIDREF(_partSlide) AND __ISVALIDREF(_twoHand)
    AND __ISVALIDREF(_partPresentSensor) AND __ISVALIDREF(_airPressureMonitor)
    AND __ISVALIDREF(_parCfg) AND __ISVALIDREF(_outCmd) AND __ISVALIDREF(_startLatched)
    AND _loadPosition.Setup(Host := Host, PressRam := PressRam, Door := Door, PartSlide := PartSlide);
END_METHOD

// §6.8 - the chain's own state on a restart (the base resets the flow state).
METHOD PROTECTED OnChainReset
// A chart restart abandons whatever the cycle was holding: the part record is
// closed by N215/N999, never by a restart, so both trackers start clean.
_partDispositioned := FALSE;
_partInMachine := FALSE;
END_METHOD

END_FUNCTION_BLOCK

// ---- 01_PneumaticPress/Release/FB_PressDemoRelease.TcPOU
// Project-owned release engineering for the pneumatic press.
// This FB is not a Fraktal module: it exposes named condition state and fills
// the Unit's authoritative release reports without adding an OPC UA tree node.
FUNCTION_BLOCK FB_PressDemoRelease EXTENDS FB_PressDemoReleaseState
VAR
    _ramExtendOk : BOOL;
    _ramExtendKey : STRING(255);
END_VAR

; // Evaluated explicitly by the owning Unit after child cyclic status is available.

METHOD Setup : BOOL
VAR_INPUT
    UnitPath : STRING(255);
END_VAR
_unitPath := UnitPath;
Setup := ModeStart.Define(Index := 1, Description := 'project.condition.airPressureOk',
    Reason := E_Reason.PERMISSIVE_NOT_MET, Bypassable := FALSE);
END_METHOD

METHOD M_Evaluate
VAR_INPUT
    PressRam : REFERENCE TO FB_CylinderCM;
    Door : REFERENCE TO FB_CylinderCM;
    PartSlide : REFERENCE TO FB_CylinderCM;
    TwoHand : REFERENCE TO FB_TwoHandStartCM;
    PneumaticPower : REFERENCE TO FB_PowerGroupCM;
    AirPressure : REFERENCE TO FB_AirPressureMonitorCM;
END_VAR
// Direction-specific functional collision prevention. Certified safety remains
// authoritative for hazardous-motion permission and safe output removal.
Door.SetDirectionalPermits(
    ExtendOk := PartSlide.OutImm.Extended AND NOT PartSlide.OutImm.Retracted
        AND NOT PartSlide.Busy AND NOT PartSlide.Error,
    RetractOk := TRUE,
    ExtendDescriptionKey := 'project.interlock.doorCloseRequiresSlideInside',
    RetractDescriptionKey := 'project.interlock.doorOpenPermitted');
PartSlide.SetDirectionalPermits(
    ExtendOk := Door.OutImm.Retracted AND NOT Door.OutImm.Extended
        AND NOT Door.Busy AND NOT Door.Error,
    RetractOk := Door.OutImm.Retracted AND NOT Door.OutImm.Extended
        AND NOT Door.Busy AND NOT Door.Error,
    ExtendDescriptionKey := 'project.interlock.slideMoveRequiresDoorOpen',
    RetractDescriptionKey := 'project.interlock.slideOutsideRequiresDoorOpen');
// Evaluate each ram-extend condition by name, then report the FIRST one that is
// missing (Core Sec.6.9 first-out). SetDirectionalPermits carries one key per
// direction, so the first-out choice is made here rather than losing it.
RamGuardClosed    := Door.OutImm.Extended AND NOT Door.OutImm.Retracted;
RamSlideInside    := PartSlide.OutImm.Extended AND NOT PartSlide.OutImm.Retracted;
RamDevicesHealthy := NOT Door.Error AND NOT PartSlide.Error;
RamAirPressureOk  := AirPressure.OutImm.PressureOk;
RamTwoHandHeld    := TwoHand.OutImm.SafeActive;
RamControlPowerOn := PneumaticPower.OutCmd.PowerOn;
_ramExtendOk := RamGuardClosed AND RamSlideInside AND RamDevicesHealthy
    AND RamAirPressureOk AND RamTwoHandHeld AND RamControlPowerOn;

IF NOT RamControlPowerOn THEN
    _ramExtendKey := 'project.interlock.pressRequiresControlPower';
ELSIF NOT RamAirPressureOk THEN
    _ramExtendKey := 'project.interlock.pressRequiresAirPressure';
ELSIF NOT RamGuardClosed THEN
    _ramExtendKey := 'project.interlock.pressRequiresGuardClosed';
ELSIF NOT RamSlideInside THEN
    _ramExtendKey := 'project.interlock.pressRequiresSlideInside';
ELSIF NOT RamDevicesHealthy THEN
    _ramExtendKey := 'project.interlock.pressRequiresHealthyGuardSlide';
ELSIF NOT RamTwoHandHeld THEN
    _ramExtendKey := 'project.interlock.pressRequiresTwoHandHeld';
ELSE
    _ramExtendKey := 'project.interlock.pressRamExtendPermitted';
END_IF

PressRam.SetDirectionalPermits(
    ExtendOk := _ramExtendOk,
    RetractOk := TRUE,
    ExtendDescriptionKey := _ramExtendKey,
    RetractDescriptionKey := 'project.interlock.pressRetractPermitted');

// Mode-entry release is distinct from future AUTO waits. Part presence and the
// two-hand edge remain live conditions in the AUTO SFC action.
ModeStartAirPressureOk := AirPressure.OutImm.PressureOk;
ModeStart.Cond[1] := ModeStartAirPressureOk;
ModeStart();
END_METHOD

METHOD M_AppendStart
VAR_IN_OUT
    Report : ST_ReleaseReport;
END_VAR
ModeStart.AppendFailed(SourcePath := _unitPath, Report := Report);
END_METHOD

METHOD M_AppendManual
VAR_INPUT
    TargetPath : STRING(255);
    Value : DINT;
    PressRam : REFERENCE TO FB_CylinderCM;
    Door : REFERENCE TO FB_CylinderCM;
    PartSlide : REFERENCE TO FB_CylinderCM;
END_VAR
VAR_IN_OUT
    Report : ST_ReleaseReport;
END_VAR
IF TargetPath = PressRam.Name THEN
    PressRam.AppendDirectionalRelease(Value := Value, Report := Report);
ELSIF TargetPath = Door.Name THEN
    Door.AppendDirectionalRelease(Value := Value, Report := Report);
ELSIF TargetPath = PartSlide.Name THEN
    PartSlide.AppendDirectionalRelease(Value := Value, Report := Report);
ELSE
    IF Report.Count < PL_Fraktal.MAX_RELEASE_REASONS THEN
        Report.Count := Report.Count + 1;
        Report.Reasons[Report.Count].Description := 'std.error.unsupportedManualTarget';
        Report.Reasons[Report.Count].ReasonCode := E_Reason.UNSUPPORTED_COMMAND;
        Report.Reasons[Report.Count].SourcePath := _unitPath;
        Report.Reasons[Report.Count].Kind := E_ReleaseKind.OTHER;
        Report.Reasons[Report.Count].Bypassable := FALSE;
    ELSE
        ; // bounded report is full; no array write is attempted
    END_IF
END_IF
END_METHOD

END_FUNCTION_BLOCK

// ---- 01_PneumaticPress/Release/FB_PressDemoReleaseState.TcPOU
// The state the press's two release renditions (ST FB_PressDemoRelease, LD
// FB_LD_PressDemoRelease) share. Both declared this block word for word; it is
// declared once here and each rendition keeps only its LOGIC, which is the
// part the bench exists to carry twice (§1.1 O9). Not a Fraktal module.
FUNCTION_BLOCK FB_PressDemoReleaseState
VAR_OUTPUT
    ModeStart : FB_PermIntlk;
    ModeStartAirPressureOk : BOOL;
    // Ram-extend permissive, split into individually named conditions. A single
    // composite permit could only ever report one composite key, so releasing
    // the two-hand button - the NORMAL way an operator stops a stroke - was
    // indistinguishable from a guard fault, an air loss or a power loss.
    RamGuardClosed   : BOOL;
    RamSlideInside   : BOOL;
    RamDevicesHealthy: BOOL;
    RamAirPressureOk : BOOL;
    RamTwoHandHeld   : BOOL;
    RamControlPowerOn: BOOL;
END_VAR
VAR
    _unitPath : STRING(255);
END_VAR

;

// Copy the evaluated conditions into the Unit's published record. Called for
// the SELECTED rendition only, straight after it evaluated, every scan.
METHOD M_PublishTo
VAR_IN_OUT
    Conditions : ST_PressDemoReleaseConditions;
END_VAR
Conditions.ModeStartAirPressureOk := ModeStartAirPressureOk;
Conditions.RamGuardClosed := RamGuardClosed;
Conditions.RamSlideInside := RamSlideInside;
Conditions.RamDevicesHealthy := RamDevicesHealthy;
Conditions.RamAirPressureOk := RamAirPressureOk;
Conditions.RamTwoHandHeld := RamTwoHandHeld;
Conditions.RamControlPowerOn := RamControlPowerOn;
END_METHOD

END_FUNCTION_BLOCK

// ---- 01_PneumaticPress/Release/FB_LD_PressDemoRelease.TcPOU
// Project-owned release engineering for the pneumatic press, authored in LADDER.
//
// This is an O2 DEMONSTRATION IN THE BENCH, not a per-project pattern. Core
// §6.8/§7.2 permit a sequence or an interlock to be authored in ST, SFC or LD,
// and the only way that claim is testable is to carry a rendition and compile
// it. Two renditions of one interlock is duplication §1.1 O9 would otherwise
// forbid outright - it is justified here, and ONLY here, because demonstrating
// the language choice IS this project's purpose, exactly as the three AUTO
// chain renditions are. A real project writes this once, in one language.
// FB_PressDemoUnit.RELEASE_LANGUAGE selects which one is evaluated.
//
// Same public surface as FB_PressDemoRelease so the Unit binds either without
// any other difference, and like it this is not a Fraktal module: it exposes
// named condition state and fills the Unit's authoritative release reports
// without adding an OPC UA tree node.
FUNCTION_BLOCK FB_LD_PressDemoRelease EXTENDS FB_PressDemoReleaseState
VAR
    _ramExtendOk : BOOL;
    _ramExtendKey : STRING(255);
    // AppendFailed returns the new report count. ST may discard a return value;
    // a rung has to land it somewhere, and the ENO slot is not that somewhere.
    _appendCount : INT;
END_VAR

; // Evaluated explicitly by the owning Unit after child cyclic status is available.

METHOD Setup : BOOL
VAR_INPUT
    UnitPath : STRING(255);
END_VAR
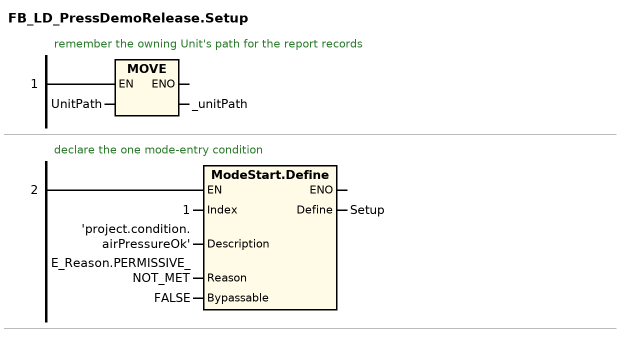
// NETWORK 1
// remember the owning Unit's path for the report records
_unitPath := UnitPath;

// NETWORK 2
// declare the one mode-entry condition
Setup := ModeStart.Define(Index := 1, Description := 'project.condition.airPressureOk', Reason := E_Reason.PERMISSIVE_NOT_MET, Bypassable := FALSE);
END_METHOD

METHOD M_Evaluate
VAR_INPUT
    PressRam : REFERENCE TO FB_CylinderCM;
    Door : REFERENCE TO FB_CylinderCM;
    PartSlide : REFERENCE TO FB_CylinderCM;
    TwoHand : REFERENCE TO FB_TwoHandStartCM;
    PneumaticPower : REFERENCE TO FB_PowerGroupCM;
    AirPressure : REFERENCE TO FB_AirPressureMonitorCM;
END_VAR
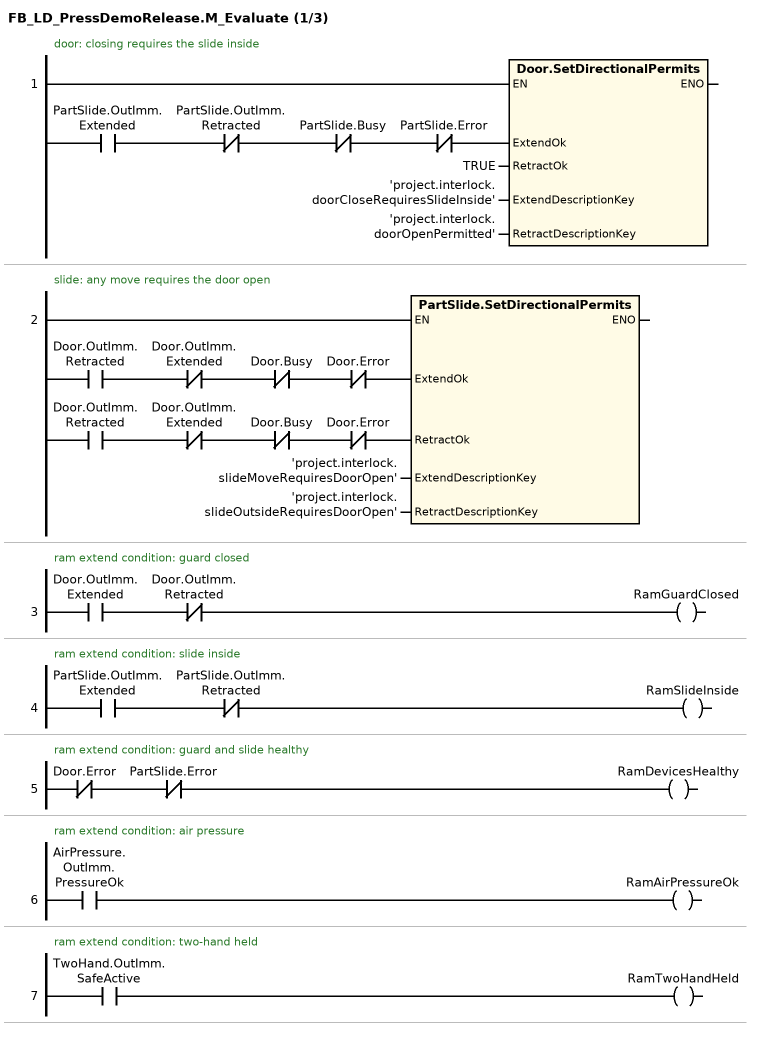
// NETWORK 1
// door: closing requires the slide inside
Door.SetDirectionalPermits(ExtendOk := PartSlide.OutImm.Extended AND NOT PartSlide.OutImm.Retracted AND NOT PartSlide.Busy AND NOT PartSlide.Error, RetractOk := TRUE, ExtendDescriptionKey := 'project.interlock.doorCloseRequiresSlideInside', RetractDescriptionKey := 'project.interlock.doorOpenPermitted');

// NETWORK 2
// slide: any move requires the door open
PartSlide.SetDirectionalPermits(ExtendOk := Door.OutImm.Retracted AND NOT Door.OutImm.Extended AND NOT Door.Busy AND NOT Door.Error, RetractOk := Door.OutImm.Retracted AND NOT Door.OutImm.Extended AND NOT Door.Busy AND NOT Door.Error, ExtendDescriptionKey := 'project.interlock.slideMoveRequiresDoorOpen', RetractDescriptionKey := 'project.interlock.slideOutsideRequiresDoorOpen');

// NETWORK 3
// ram extend condition: guard closed
RamGuardClosed := Door.OutImm.Extended AND NOT Door.OutImm.Retracted;

// NETWORK 4
// ram extend condition: slide inside
RamSlideInside := PartSlide.OutImm.Extended AND NOT PartSlide.OutImm.Retracted;

// NETWORK 5
// ram extend condition: guard and slide healthy
RamDevicesHealthy := NOT Door.Error AND NOT PartSlide.Error;

// NETWORK 6
// ram extend condition: air pressure
RamAirPressureOk := AirPressure.OutImm.PressureOk;

// NETWORK 7
// ram extend condition: two-hand held
RamTwoHandHeld := TwoHand.OutImm.SafeActive;

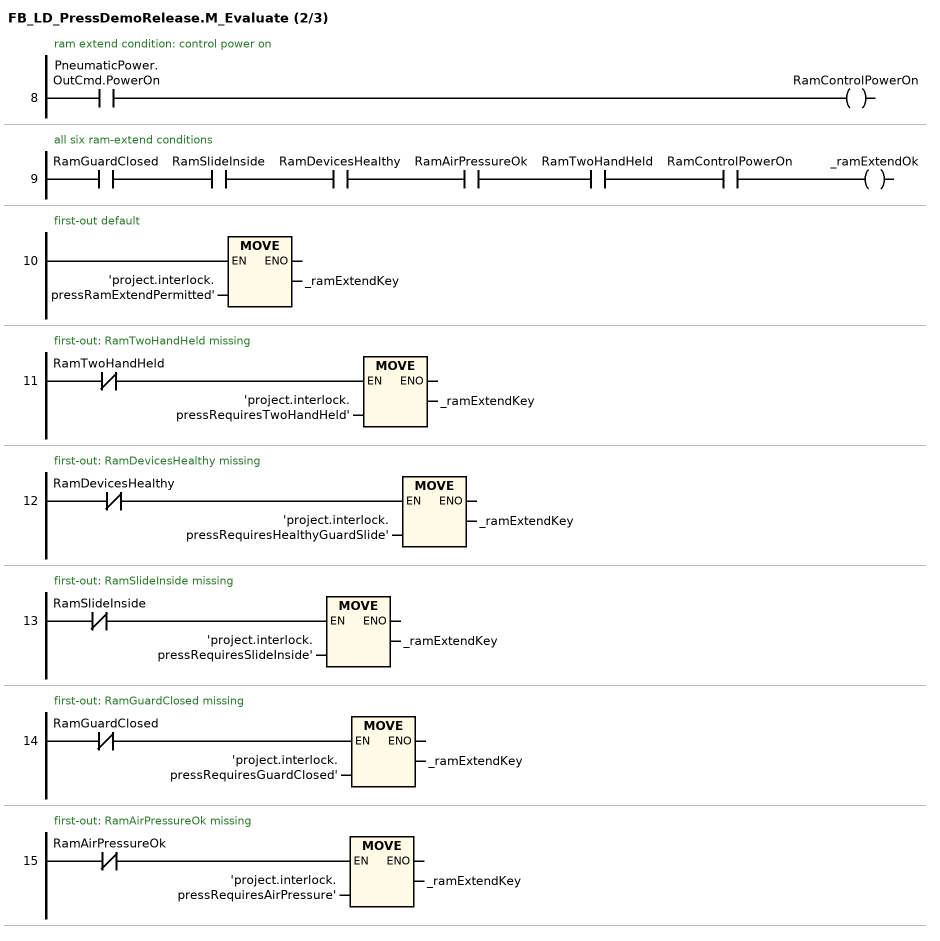
// NETWORK 8
// ram extend condition: control power on
RamControlPowerOn := PneumaticPower.OutCmd.PowerOn;

// NETWORK 9
// all six ram-extend conditions
_ramExtendOk := RamGuardClosed AND RamSlideInside AND RamDevicesHealthy AND RamAirPressureOk AND RamTwoHandHeld AND RamControlPowerOn;

// NETWORK 10
// first-out default
_ramExtendKey := 'project.interlock.pressRamExtendPermitted';

// NETWORK 11
// first-out: RamTwoHandHeld missing
IF NOT RamTwoHandHeld THEN _ramExtendKey := 'project.interlock.pressRequiresTwoHandHeld'; END_IF

// NETWORK 12
// first-out: RamDevicesHealthy missing
IF NOT RamDevicesHealthy THEN _ramExtendKey := 'project.interlock.pressRequiresHealthyGuardSlide'; END_IF

// NETWORK 13
// first-out: RamSlideInside missing
IF NOT RamSlideInside THEN _ramExtendKey := 'project.interlock.pressRequiresSlideInside'; END_IF

// NETWORK 14
// first-out: RamGuardClosed missing
IF NOT RamGuardClosed THEN _ramExtendKey := 'project.interlock.pressRequiresGuardClosed'; END_IF

// NETWORK 15
// first-out: RamAirPressureOk missing
IF NOT RamAirPressureOk THEN _ramExtendKey := 'project.interlock.pressRequiresAirPressure'; END_IF

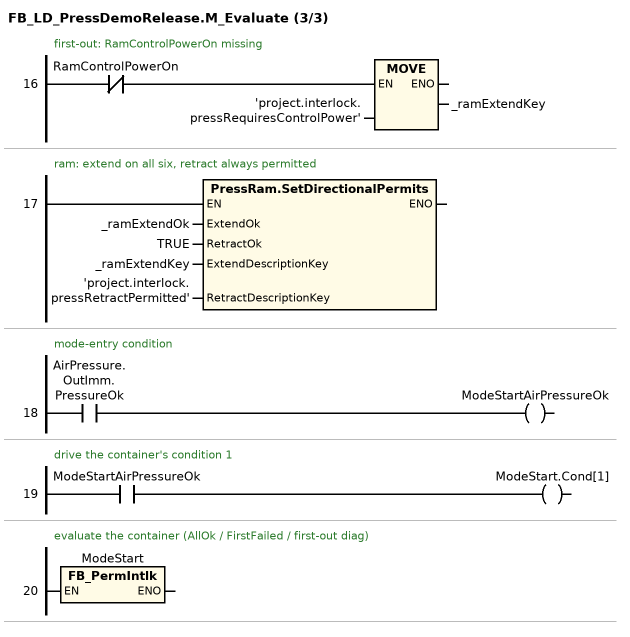
// NETWORK 16
// first-out: RamControlPowerOn missing
IF NOT RamControlPowerOn THEN _ramExtendKey := 'project.interlock.pressRequiresControlPower'; END_IF

// NETWORK 17
// ram: extend on all six, retract always permitted
PressRam.SetDirectionalPermits(ExtendOk := _ramExtendOk, RetractOk := TRUE, ExtendDescriptionKey := _ramExtendKey, RetractDescriptionKey := 'project.interlock.pressRetractPermitted');

// NETWORK 18
// mode-entry condition
ModeStartAirPressureOk := AirPressure.OutImm.PressureOk;

// NETWORK 19
// drive the container's condition 1
ModeStart.Cond[1] := ModeStartAirPressureOk;

// NETWORK 20
// evaluate the container (AllOk / FirstFailed / first-out diag)
ModeStart(); // FB_PermIntlk
END_METHOD

METHOD M_AppendStart
VAR_IN_OUT
    Report : ST_ReleaseReport;
END_VAR
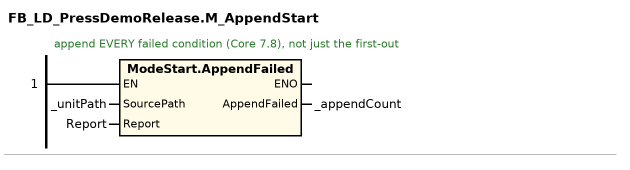
// NETWORK 1
// append EVERY failed condition (Core 7.8), not just the first-out
_appendCount := ModeStart.AppendFailed(SourcePath := _unitPath, Report := Report);
END_METHOD

// Deliberately ST, in a POU whose interlocks are ladder. This method is TARGET
// DISPATCH and bounded-report bookkeeping - matching a path against three child
// names and, failing that, writing five fields of one report row. None of that
// is condition logic, which is what O2's choice of language is about, and a
// ladder rendition of it would be longer, harder to read and no more
// demonstrative. Per-method language choice is exactly what TwinCAT offers.
METHOD M_AppendManual
VAR_INPUT
    TargetPath : STRING(255);
    Value : DINT;
    PressRam : REFERENCE TO FB_CylinderCM;
    Door : REFERENCE TO FB_CylinderCM;
    PartSlide : REFERENCE TO FB_CylinderCM;
END_VAR
VAR_IN_OUT
    Report : ST_ReleaseReport;
END_VAR
IF TargetPath = PressRam.Name THEN
    PressRam.AppendDirectionalRelease(Value := Value, Report := Report);
ELSIF TargetPath = Door.Name THEN
    Door.AppendDirectionalRelease(Value := Value, Report := Report);
ELSIF TargetPath = PartSlide.Name THEN
    PartSlide.AppendDirectionalRelease(Value := Value, Report := Report);
ELSE
    IF Report.Count < PL_Fraktal.MAX_RELEASE_REASONS THEN
        Report.Count := Report.Count + 1;
        Report.Reasons[Report.Count].Description := 'std.error.unsupportedManualTarget';
        Report.Reasons[Report.Count].ReasonCode := E_Reason.UNSUPPORTED_COMMAND;
        Report.Reasons[Report.Count].SourcePath := _unitPath;
        Report.Reasons[Report.Count].Kind := E_ReleaseKind.OTHER;
        Report.Reasons[Report.Count].Bypassable := FALSE;
    ELSE
        ; // bounded report is full; no array write is attempted
    END_IF
END_IF
END_METHOD

END_FUNCTION_BLOCK

// ---- 00_System/FB_PressIoDriver.TcPOU
// Project Hardware Driver layer. This is the only POU that accesses GVL_PressIO.
// It maps raw process-image symbols to semantic HALs and refreshes the Core
// topology publisher. It contains no sequence, mode, recipe or device behavior.
FUNCTION_BLOCK FB_PressIoDriver
VAR_OUTPUT
    // Raw N54 D2 operator buttons, republished so MAIN can drive Control On/Off
    // from hardware without becoming a second GVL_PressIO consumer.
    ControlOnButton  : BOOL;
    ControlOffButton : BOOL;
END_VAR
VAR
    _publisher : FB_IoTopologyPublisher;
    {attribute 'OPC.UA.DA' := '0'}
    _unit : REFERENCE TO FB_PressDemoUnit;
    _attached : BOOL;
    // Hardware Control-On adapter: reconstructs the safety-status mirrors from
    // the raw relay/sensor process image on a machine with a hardwired N54 D2
    // Control On circuit (no TwinSAFE controller). Status only; not a safety fn.
    _controlOn : FB_PressControlOnCircuit;
    // Reads the REAL EtherCAT slave states from the master and publishes each
    // node's live state — the fieldbus tree reflects hardware, not Control-On.
    _busHealth : FB_EcBusHealth;
END_VAR

;

METHOD Setup : BOOL
VAR_INPUT
    UnitRef : REFERENCE TO FB_PressDemoUnit;
END_VAR
VAR
    // Left all-zero: FB_EcBusHealth auto-detects the EtherCAT master's AmsNetId,
    // so the project needs no fieldbus address and no XAE link. Assign a value
    // here only for a non-standard master (remote, or several on one PC).
    ecMasterNetId : T_AmsNetIdArr;
END_VAR
_unit REF= UnitRef;
_attached := _publisher.Setup(DataRef := GVL_PressFieldbus.Topology, ResetData := FALSE)
    AND __ISVALIDREF(_unit);
// Map the press topology to the EtherCAT master's slaves. The catalog defines
// node 1 = CX2030 master and nodes 2..6 = the five devices in the project tree
// (EK1200 coupler, EL1809, EL2809, EL6001, EL9011).
//
// Only THREE of those are slaves the master enumerates: the EK1200 coupler and
// the EL9011 end cap carry the bus but have no EtherCAT slave controller on the
// process-data ring, so they never appear in FB_EcGetAllSlaveStates. Declaring
// SlaveCount := 5 made the master's slave i land on catalog node i, shifting
// every state onto its neighbour: the EL6001's OP was published onto the
// EL2809, and the EL6001 itself read OFFLINE while it was perfectly healthy.
// State the mapping instead of assuming it.
_busHealth.Setup(Publisher := _publisher, MasterNetIdArr := ecMasterNetId,
    FirstSlaveNode := 3, SlaveCount := 3, MasterNodeIndex := 1);
_busHealth.M_MapSlaveNode(SlaveIndex := 1, NodeIndex := 3);   // EL1809
_busHealth.M_MapSlaveNode(SlaveIndex := 2, NodeIndex := 4);   // EL2809
_busHealth.M_MapSlaveNode(SlaveIndex := 3, NodeIndex := 5);   // EL6001
_busHealth.M_MapPassiveNode(NodeIndex := 2);                  // EK1200 coupler
_busHealth.M_MapPassiveNode(NodeIndex := 6);                  // EL9011 end cap
Setup := _attached;
END_METHOD

METHOD M_ReadInputs
VAR_IN_OUT
    PressHal : ST_CylinderHal;
    DoorHal : ST_CylinderHal;
    SlideHal : ST_CylinderHal;
    TwoHandHal : ST_TwoHandHal;
    PowerHal : ST_PowerGroupHal;
    PartPresentHal : ST_DigitalInputHal;
    AirPressureHal : ST_AirPressureHal;
    RawEStopHealthy : BOOL;
    SafeEStopOk : BOOL;
    SafeGuardClosed : BOOL;
    SafeTwoHandActive : BOOL;
    SafePneumaticPermit : BOOL;
    SafetyFieldbusHealthy : BOOL;
    StandardIoHealthy : BOOL;
END_VAR
VAR
    // EtherCAT process-image validity, DETECTED from the fieldbus master by the
    // library (FB_EcBusHealth) — the project no longer declares/links a RealBusOk.
    busOk : BOOL;
END_VAR
busOk := _busHealth.M_BusOk();
// Physical feeder retracted = logical slide inside; extended = outside.
SlideHal.ExtendedFb := GVL_PressIO._101B301A;
SlideHal.RetractedFb := GVL_PressIO._101B301B;
DoorHal.ExtendedFb := GVL_PressIO._101B201A;
DoorHal.RetractedFb := GVL_PressIO._101B201B;
PressHal.ExtendedFb := GVL_PressIO._101B202A;
PressHal.RetractedFb := GVL_PressIO._101B202B;
TwoHandHal.RightPressed := GVL_PressIO._101S101;
TwoHandHal.LeftPressed := GVL_PressIO._101S102;
PartPresentHal.Value := GVL_PressIO._101B601;
AirPressureHal.LowPressure := GVL_PressIO._000MB085A_2;
AirPressureHal.OperatingPressure := GVL_PressIO._000MB085A_4;
PowerHal.PowerFeedback := GVL_PressIO._000K911_Y32;
// This machine's safety is a hardwired N54 D2 Control On relay chain, not a
// TwinSAFE controller, so the GVL_PressSafety AT %I* aliases are never written.
// Reconstruct the read-only safety-status mirrors from the raw relay/sensor
// process image via the Control-On adapter. The relay chain remains the safety
// authority; these values drive HMI/interlock display only.
_controlOn.M_Evaluate(
    // POLARITY: =000+S1-K910A:14 is "Emergency Switch 1 PRESSED" (N54 D2), and on
    // THIS machine the contact is CONFIRMED NORMALLY OPEN - not pressed reads
    // FALSE, pressed reads TRUE - so inverting it yields the "healthy" mirror
    // this adapter publishes. Read un-inverted, a healthy machine reported
    // E-stop-unhealthy and control power was withheld (POWER_ENABLE_WITHHELD)
    // even with the relay chain demonstrably closed.
    //
    // DEMO WIRING ONLY - NOT FAIL-SAFE. A normally-open E-stop contact cannot
    // distinguish "not pressed" from a broken wire, a pulled terminal or a dead
    // input card: all read FALSE, and this mirror would then report HEALTHY.
    // ISO 13850 / EN 60204-1 require a normally-CLOSED contact so that any break
    // forces the stop. A production machine must rewire to NC and drop this
    // inversion. This mirror is diagnostic only - the hardwired relay chain
    // remains the safety authority (Core Sec.9), which is what keeps the
    // non-fail-safe wiring tolerable on a demo rig and nowhere else.
    EStopHealthyMirror := NOT GVL_PressIO._000K910A,
    DoorClosed := GVL_PressIO._101B201A,
    LeftButton := GVL_PressIO._101S102,
    RightButton := GVL_PressIO._101S101,
    ControlOnFeedback := GVL_PressIO._000K911_Y32,
    BusOk := busOk,
    ControlOnButton := GVL_PressIO._000BS901,
    ControlOffButton := GVL_PressIO._000BS902,
    AirPressureOk := GVL_PressIO._000MB085A_4 AND NOT GVL_PressIO._000MB085A_2);
RawEStopHealthy := _controlOn.RawEStopHealthy;
SafeEStopOk := _controlOn.SafeEStopOk;
SafeGuardClosed := _controlOn.SafeGuardClosed;
SafeTwoHandActive := _controlOn.SafeTwoHandActive;
SafePneumaticPermit := _controlOn.SafePneumaticPermit;
SafetyFieldbusHealthy := _controlOn.SafetyFieldbusHealthy;
StandardIoHealthy := _controlOn.StandardIoHealthy;
PartPresentHal.Quality := StandardIoHealthy;
AirPressureHal.Quality := StandardIoHealthy;
ControlOnButton := GVL_PressIO._000BS901;
ControlOffButton := GVL_PressIO._000BS902;
END_METHOD

// Also withdraws every held §10.5.1 force: under USE_SIMULATION no physical
// output is driven at all, so a set-point armed earlier must not survive here
// and reappear the moment a real write path runs (§10.5.1 rule 3).
METHOD M_ClearOutputs
_publisher.M_ApplyForces(Enabled := FALSE);
GVL_PressIO._101K301A := FALSE; GVL_PressIO._101K301B := FALSE;
GVL_PressIO._101K201A := FALSE; GVL_PressIO._101K201B := FALSE;
GVL_PressIO._101K202A := FALSE; GVL_PressIO._101K202B := FALSE;
GVL_PressIO._101P101 := FALSE; GVL_PressIO._101P102 := FALSE;
GVL_PressIO._000K951_A1 := FALSE; GVL_PressIO._000K911_A1 := FALSE;
END_METHOD

METHOD M_WriteOutputs
VAR_INPUT
    PressHal : ST_CylinderHal;
    DoorHal : ST_CylinderHal;
    SlideHal : ST_CylinderHal;
    PowerHal : ST_PowerGroupHal;
    LampsOn : BOOL;
    ControlCircuitMappingConfirmed : BOOL;
    // Core §10.5.1 rule 3 - FB_UnitBase.M_ForcePermitted() of the owning Unit.
    // The SAME predicate its ForceChannel accepted the request with, so a force
    // can never be accepted under conditions in which it would not be applied,
    // and leaving idle MANUAL withdraws every held set-point on that scan.
    ForcePermitted : BOOL;
END_VAR
// One call decides whether held set-points apply this scan, and withdraws them
// all on the falling edge. It runs BEFORE the writes below, so the very scan
// the Unit leaves idle MANUAL is already driven by application logic again.
_publisher.M_ApplyForces(Enabled := ForcePermitted);
// M_EffectiveBool returns the value, so each line still reads as the plain
// assignment it was: the application value, or the held force set-point while
// forcing is permitted and this channel is forced.
GVL_PressIO._101K301A := _publisher.M_EffectiveBool(NodeIndex := 4, ChannelIndex := 1, Value := SlideHal.ExtendOut);
GVL_PressIO._101K301B := _publisher.M_EffectiveBool(NodeIndex := 4, ChannelIndex := 2, Value := SlideHal.RetractOut);
GVL_PressIO._101K201A := _publisher.M_EffectiveBool(NodeIndex := 4, ChannelIndex := 3, Value := DoorHal.ExtendOut);
GVL_PressIO._101K201B := _publisher.M_EffectiveBool(NodeIndex := 4, ChannelIndex := 4, Value := DoorHal.RetractOut);
GVL_PressIO._101K202A := _publisher.M_EffectiveBool(NodeIndex := 4, ChannelIndex := 5, Value := PressHal.ExtendOut);
GVL_PressIO._101K202B := _publisher.M_EffectiveBool(NodeIndex := 4, ChannelIndex := 6, Value := PressHal.RetractOut);
GVL_PressIO._101P101 := _publisher.M_EffectiveBool(NodeIndex := 4, ChannelIndex := 7, Value := LampsOn);
GVL_PressIO._101P102 := _publisher.M_EffectiveBool(NodeIndex := 4, ChannelIndex := 8, Value := LampsOn);
// Ch9/Ch10 (_000K951_A1 / _000K911_A1) are never routed through the force
// path: they drive the hardwired N54 D2 Control On relay chain and the
// catalog never marks them forceable (§10.5.1 rule 4).
IF ControlCircuitMappingConfirmed THEN
    // N54 D2: these are DIFFERENT signals. SwitchControlOn is the momentary
    // button coil (2 s pulse); EnableControlOn is the bus/air permissive that
    // must be TRUE whenever the machine is healthy. Driving both from one power
    // request was why the control circuit could never energize.
    GVL_PressIO._000K951_A1 := _controlOn.SwitchControlOn;
    GVL_PressIO._000K911_A1 := _controlOn.EnableControlOn;
ELSE
    GVL_PressIO._000K951_A1 := FALSE;
    GVL_PressIO._000K911_A1 := FALSE;
END_IF
END_METHOD

// The EtherCAT adapter this driver owns, handed once to the health probe by the
// composition root (§8.12/§10.5): one master, sampled once, read by both.
METHOD M_BusHealth : POINTER TO FB_EcBusHealth
M_BusHealth := ADR(_busHealth);
END_METHOD

// Node state now comes from the REAL EtherCAT master (FB_EcBusHealth), NOT from
// the Control-On / StandardIoHealthy verdict — the HMI fieldbus tree mirrors
// the actual bus (as XAE shows it). StandardIoHealthy is no longer an input.
METHOD M_RefreshFieldbus
VAR_INPUT
    // §10.5.1: the bus picture is a diagnostic surface, so the master is only
    // scanned while a consumer is actually reading it (the HMI fieldbus view is
    // open). Pass FALSE to park the scan; published states are then held, not
    // invalidated. One scan always runs after Setup so M_BusOk() has real data.
    BusViewActive : BOOL;
END_VAR
VAR
    D : ST_Diagnostic;
END_VAR
IF _attached THEN
    _busHealth.M_RequestScan(Active := BusViewActive);
    _busHealth.M_Refresh();  // publishes each node's real INIT/PREOP/SAFEOP/OP/FAULT
    _publisher.M_SetDigitalValue(NodeIndex := 3, ChannelIndex := 1, Value := GVL_PressIO._101B301A);
    _publisher.M_SetDigitalValue(NodeIndex := 3, ChannelIndex := 2, Value := GVL_PressIO._101B301B);
    _publisher.M_SetDigitalValue(NodeIndex := 3, ChannelIndex := 3, Value := GVL_PressIO._101B201A);
    _publisher.M_SetDigitalValue(NodeIndex := 3, ChannelIndex := 4, Value := GVL_PressIO._101B201B);
    _publisher.M_SetDigitalValue(NodeIndex := 3, ChannelIndex := 5, Value := GVL_PressIO._101B202A);
    _publisher.M_SetDigitalValue(NodeIndex := 3, ChannelIndex := 6, Value := GVL_PressIO._101B202B);
    _publisher.M_SetDigitalValue(NodeIndex := 3, ChannelIndex := 7, Value := GVL_PressIO._101S101);
    _publisher.M_SetDigitalValue(NodeIndex := 3, ChannelIndex := 8, Value := GVL_PressIO._101S102);
    _publisher.M_SetDigitalValue(NodeIndex := 3, ChannelIndex := 9, Value := GVL_PressIO._000MB085A_2);
    _publisher.M_SetDigitalValue(NodeIndex := 3, ChannelIndex := 10, Value := GVL_PressIO._000MB085A_4);
    _publisher.M_SetDigitalValue(NodeIndex := 3, ChannelIndex := 11, Value := GVL_PressIO._101B601);
    _publisher.M_SetDigitalValue(NodeIndex := 3, ChannelIndex := 12, Value := GVL_PressIO._000K911_Y32);
    _publisher.M_SetDigitalValue(NodeIndex := 3, ChannelIndex := 13, Value := GVL_PressIO._000K910A);
    _publisher.M_SetDigitalValue(NodeIndex := 4, ChannelIndex := 1, Value := GVL_PressIO._101K301A);
    _publisher.M_SetDigitalValue(NodeIndex := 4, ChannelIndex := 2, Value := GVL_PressIO._101K301B);
    _publisher.M_SetDigitalValue(NodeIndex := 4, ChannelIndex := 3, Value := GVL_PressIO._101K201A);
    _publisher.M_SetDigitalValue(NodeIndex := 4, ChannelIndex := 4, Value := GVL_PressIO._101K201B);
    _publisher.M_SetDigitalValue(NodeIndex := 4, ChannelIndex := 5, Value := GVL_PressIO._101K202A);
    _publisher.M_SetDigitalValue(NodeIndex := 4, ChannelIndex := 6, Value := GVL_PressIO._101K202B);
    _publisher.M_SetDigitalValue(NodeIndex := 4, ChannelIndex := 7, Value := GVL_PressIO._101P101);
    _publisher.M_SetDigitalValue(NodeIndex := 4, ChannelIndex := 8, Value := GVL_PressIO._101P102);
    _publisher.M_SetDigitalValue(NodeIndex := 4, ChannelIndex := 9, Value := GVL_PressIO._000K951_A1);
    _publisher.M_SetDigitalValue(NodeIndex := 4, ChannelIndex := 10, Value := GVL_PressIO._000K911_A1);
    _publisher.M_BeginDiagnosticRefresh();
    D := _unit.PressRam.Status.Diagnostic;
    _M_ApplyCylinderDiagnostic(Diagnostic := D,
        ExtendedTag := _unit.PressRam.OutImm.ExtendedSensorTag,
        RetractedTag := _unit.PressRam.OutImm.RetractedSensorTag);
    D := _unit.Door.Status.Diagnostic;
    _M_ApplyCylinderDiagnostic(Diagnostic := D,
        ExtendedTag := _unit.Door.OutImm.ExtendedSensorTag,
        RetractedTag := _unit.Door.OutImm.RetractedSensorTag);
    D := _unit.PartSlide.Status.Diagnostic;
    _M_ApplyCylinderDiagnostic(Diagnostic := D,
        ExtendedTag := _unit.PartSlide.OutImm.ExtendedSensorTag,
        RetractedTag := _unit.PartSlide.OutImm.RetractedSensorTag);
    D := _unit.AirPressureMonitor.Status.Diagnostic;
    _publisher.M_ApplyDiagnostic(Diagnostic := D);
    IF TO_DINT(D.ReasonCode) = PL_ModuleReasons.AIR_SWITCH_CONFLICT THEN
        _publisher.M_ApplyDiagnosticToTag(Diagnostic := D,
            Tag := _unit.AirPressureMonitor.OutImm.LowSensorTag);
        _publisher.M_ApplyDiagnosticToTag(Diagnostic := D,
            Tag := _unit.AirPressureMonitor.OutImm.OperatingSensorTag);
    ELSE
        ;
    END_IF
    // §10.5.1 — the RS232 terminal's process image, published like any other
    // channel so a dead serial link is visible on the bus page instead of invisible.
    _publisher.M_SetAnalogValue(NodeIndex := 5, ChannelIndex := 1, Value := USINT_TO_REAL(GVL_PressIO._000K010D1_Status));
    _publisher.M_SetAnalogValue(NodeIndex := 5, ChannelIndex := 2, Value := USINT_TO_REAL(GVL_PressIO._000K010D1_DataIn0));
    _publisher.M_SetAnalogValue(NodeIndex := 5, ChannelIndex := 3, Value := USINT_TO_REAL(GVL_PressIO._000K010D1_DataIn1));
    _publisher.M_SetAnalogValue(NodeIndex := 5, ChannelIndex := 4, Value := USINT_TO_REAL(GVL_PressIO._000K010D1_DataIn2));
    _publisher.M_SetAnalogValue(NodeIndex := 5, ChannelIndex := 5, Value := USINT_TO_REAL(GVL_PressIO._000K010D1_Ctrl));
    _publisher.M_SetAnalogValue(NodeIndex := 5, ChannelIndex := 6, Value := USINT_TO_REAL(GVL_PressIO._000K010D1_DataOut0));
    _publisher.M_SetAnalogValue(NodeIndex := 5, ChannelIndex := 7, Value := USINT_TO_REAL(GVL_PressIO._000K010D1_DataOut1));
    _publisher.M_SetAnalogValue(NodeIndex := 5, ChannelIndex := 8, Value := USINT_TO_REAL(GVL_PressIO._000K010D1_DataOut2));
    _publisher.M_ApplyDiagnostic(Diagnostic := _unit.Status.Diagnostic);
ELSE
    ;
END_IF
END_METHOD

METHOD PRIVATE _M_ApplyCylinderDiagnostic
VAR_INPUT
    Diagnostic : ST_Diagnostic;
    ExtendedTag : STRING(80);
    RetractedTag : STRING(80);
END_VAR
_publisher.M_ApplyDiagnostic(Diagnostic := Diagnostic);
IF TO_DINT(Diagnostic.ReasonCode) = PL_ModuleReasons.CYL_BOTH_SENSORS THEN
    _publisher.M_ApplyDiagnosticToTag(Diagnostic := Diagnostic, Tag := ExtendedTag);
    _publisher.M_ApplyDiagnosticToTag(Diagnostic := Diagnostic, Tag := RetractedTag);
ELSE
    ;
END_IF
END_METHOD

END_FUNCTION_BLOCK

// ---- 00_System/FB_PressControlOnCircuit.TcPOU
// Hardware Control-On adapter for a machine whose safety is a HARDWIRED relay
// chain (Bosch/Nexeed N54 D2 "Control On", Pilz-style), NOT a TwinSAFE
// controller. The standard PLC is not a safety function here: the relay circuit
// remains the safety authority. This adapter only RECONSTRUCTS the read-only
// GVL_PressSafety-equivalent status the rest of the application expects, from the
// ordinary process-image inputs and the relay-chain Control On feedback, so the
// HMI and interlocks reflect the real machine instead of failing closed on
// unlinked TwinSAFE aliases.
//
// It produces status only (no safe outputs). The functional EnableControlOn /
// SwitchControlOn requests to the relay chain are driven by the existing power
// group -> FB_PressIoDriver.M_WriteOutputs path, gated by
// ControlCircuitMappingConfirmed until the electrical semantics are confirmed.
FUNCTION_BLOCK FB_PressControlOnCircuit
VAR_OUTPUT
    // Read-only mirrors, matching the six GVL_PressSafety aliases + the raw
    // E-stop mirror the driver forwards. TRUE = healthy/safe/present.
    RawEStopHealthy       : BOOL;
    SafeEStopOk           : BOOL;
    SafeGuardClosed       : BOOL;
    SafeTwoHandActive     : BOOL;
    SafePneumaticPermit   : BOOL;
    SafetyFieldbusHealthy : BOOL;
    StandardIoHealthy     : BOOL;

    // --- N54 D2 functional requests to the relay chain (not safety outputs) ---
    // EnableControlOn is a PERMISSIVE, not a command: per the standard it is set
    // at the start of the cycle from "bus OK and control-off not pressed", and
    // reset by the Main/Safety-Valve add-ons when compressed-air monitoring
    // errors. It must NOT wait for an operator power request, which is why the
    // control circuit could never be energized headless.
    EnableControlOn : BOOL;
    // SwitchControlOn is the BUTTON coil: TRUE for exactly two seconds on the
    // rising edge of the Control On button, however long the button is held, so
    // the guard doors have time to lock. Control Off has priority and cancels it.
    SwitchControlOn : BOOL;
    ControlOffSet   : BOOL;   // per the standard: NOT EnableControlOn
END_VAR
VAR
    _onEdge       : R_TRIG;
    _switchTimer  : TON;
    _switchActive : BOOL;
END_VAR

;

// Reconstruct the status mirrors from raw relay/sensor inputs. All inputs are
// ordinary (non-safety-rated) process-image values; the relay chain owns the
// actual safety function. Called once per scan by FB_PressIoDriver, the sole
// GVL_PressIO consumer.
METHOD M_Evaluate
VAR_INPUT
    EStopHealthyMirror : BOOL; // _000K910A: ordinary E-stop-healthy mirror
    DoorClosed         : BOOL; // _101B201A: guard-door closed sensor
    LeftButton         : BOOL; // _101S102: left two-hand raw button
    RightButton        : BOOL; // _101S101: right two-hand raw button
    ControlOnFeedback  : BOOL; // _000K911_Y32: relay-chain Control On established
    BusOk              : BOOL; // EtherCAT process image valid (link master OP state)
    ControlOnButton    : BOOL; // _000BS901: IsControlOnButtonPressed
    ControlOffButton   : BOOL; // _000BS902: IsControlOffButtonPressed
    AirPressureOk      : BOOL; // compressed-air monitoring OK (Main/Safety Valve)
END_VAR
// Fieldbus health: the standard and (functional) safety I/O share one EtherCAT
// segment on this machine, so both mirror the bus-valid signal.
StandardIoHealthy     := BusOk;
SafetyFieldbusHealthy := BusOk;

// E-stop: the ordinary healthy mirror gated by a valid process image. This is a
// diagnostic mirror of the relay-chain E-stop, not an evaluated safe result.
RawEStopHealthy := EStopHealthyMirror;
SafeEStopOk     := EStopHealthyMirror AND BusOk;

// Guard: the door-closed sensor. Plausibility (per N54 D2 Safety Door add-on) is
// enforced in the relay chain; here it is the single available door signal.
SafeGuardClosed := DoorClosed AND BusOk;

// Two-hand: functional (both raw buttons) with E-stop healthy. The safety-rated
// two-hand evaluation lives in the relay chain; this drives interlock/HMI only.
SafeTwoHandActive := LeftButton AND RightButton AND SafeEStopOk AND BusOk;

// Pneumatic permit: the relay-chain Control On feedback IS the enabled state.
// Per N54 D2 the Main/Safety Valve add-ons already reset EnableControlOn on a
// compressed-air error and the Safety Door add-on on a guard error, so the
// K911_Y32 feedback subsumes air + guard monitoring. Gate on E-stop for defense
// in depth (the air-pressure inputs are read separately by the air HAL).
SafePneumaticPermit := ControlOnFeedback AND SafeEStopOk;

